//PR1006_REV_002685_TIMTRO
GVL.EF.S_Fus_1_01						:= GVL.IIVD.X_Fus_0_D1.v AND _FB_CanRx_Message_Unpack_261.S_Bit_6;
GVL.EF.S_Fus_1_02						:= GVL.IIVD.X_Fus_0_D1.v AND _FB_CanRx_Message_Unpack_261.S_Bit_4;
GVL.EF.S_Fus_1_03						:= GVL.IIVD.X_Fus_0_D1.v AND _FB_CanRx_Message_Unpack_261.S_Bit_2;
GVL.EF.S_Fus_1_04						:= GVL.IIVD.X_Fus_0_D1.v AND _FB_CanRx_Message_Unpack_261.S_Bit_0;	 
GVL.EF.S_Fus_1_05						:= GVL.IIVD.X_Fus_0_D2.v AND _FB_CanRx_Message_Unpack_261.S_Bit_14;
GVL.EF.S_Fus_1_06						:= GVL.IIVD.X_Fus_0_D2.v AND _FB_CanRx_Message_Unpack_261.S_Bit_12;
GVL.EF.S_Fus_1_07						:= GVL.IIVD.X_Fus_0_D2.v AND _FB_CanRx_Message_Unpack_261.S_Bit_10;
GVL.EF.S_Fus_1_08						:= GVL.IIVD.X_Fus_0_D2.v AND _FB_CanRx_Message_Unpack_261.S_Bit_8;					
GVL.EF.S_Fus_1_09						:= GVL.IIVD.X_Fus_0_D3.v AND _FB_CanRx_Message_Unpack_261.S_Bit_22;
GVL.EF.S_Fus_1_10						:= GVL.IIVD.X_Fus_0_D3.v AND _FB_CanRx_Message_Unpack_261.S_Bit_20;
GVL.EF.S_Fus_1_11						:= GVL.IIVD.X_Fus_0_D3.v AND _FB_CanRx_Message_Unpack_261.S_Bit_18;
GVL.EF.S_Fus_1_12						:= GVL.IIVD.X_Fus_0_D3.v AND _FB_CanRx_Message_Unpack_261.S_Bit_16;							  
GVL.EF.S_Fus_1_13						:= GVL.IIVD.X_Fus_0_D4.v AND _FB_CanRx_Message_Unpack_261.S_Bit_30;
GVL.EF.S_Fus_1_14						:= GVL.IIVD.X_Fus_0_D4.v AND _FB_CanRx_Message_Unpack_261.S_Bit_28;
GVL.EF.S_Fus_1_15						:= GVL.IIVD.X_Fus_0_D4.v AND _FB_CanRx_Message_Unpack_261.S_Bit_26;
GVL.EF.S_Fus_1_16						:= GVL.IIVD.X_Fus_0_D4.v AND _FB_CanRx_Message_Unpack_261.S_Bit_24;										
GVL.EF.S_Fus_1_17						:= GVL.IIVD.X_Fus_0_D5.v AND _FB_CanRx_Message_Unpack_261.S_Bit_38;
GVL.EF.S_Fus_1_18						:= GVL.IIVD.X_Fus_0_D5.v AND _FB_CanRx_Message_Unpack_261.S_Bit_36;
GVL.EF.S_Fus_1_19						:= GVL.IIVD.X_Fus_0_D5.v AND _FB_CanRx_Message_Unpack_261.S_Bit_34;
GVL.EF.S_Fus_1_20						:= GVL.IIVD.X_Fus_0_D5.v AND _FB_CanRx_Message_Unpack_261.S_Bit_32;		  
GVL.EF.S_Fus_1_21						:= GVL.IIVD.X_Fus_0_D6.v AND _FB_CanRx_Message_Unpack_261.S_Bit_46;
GVL.EF.S_Fus_1_22						:= GVL.IIVD.X_Fus_0_D6.v AND _FB_CanRx_Message_Unpack_261.S_Bit_44;
GVL.EF.S_Fus_1_23						:= GVL.IIVD.X_Fus_0_D6.v AND _FB_CanRx_Message_Unpack_261.S_Bit_42;
GVL.EF.S_Fus_1_24						:= GVL.IIVD.X_Fus_0_D6.v AND _FB_CanRx_Message_Unpack_261.S_Bit_40;		  
GVL.EF.S_Fus_1_25						:= GVL.IIVD.X_Fus_0_D7.v AND _FB_CanRx_Message_Unpack_261.S_Bit_54;
GVL.EF.S_Fus_1_26						:= GVL.IIVD.X_Fus_0_D7.v AND _FB_CanRx_Message_Unpack_261.S_Bit_52;
GVL.EF.S_Fus_1_27						:= GVL.IIVD.X_Fus_0_D7.v AND _FB_CanRx_Message_Unpack_261.S_Bit_50;
GVL.EF.S_Fus_1_28						:= GVL.IIVD.X_Fus_0_D7.v AND _FB_CanRx_Message_Unpack_261.S_Bit_48;												  
GVL.EF.S_Fus_1_29						:= GVL.IIVD.X_Fus_0_D8.v AND _FB_CanRx_Message_Unpack_261.S_Bit_62;
GVL.EF.S_Fus_1_30						:= GVL.IIVD.X_Fus_0_D8.v AND _FB_CanRx_Message_Unpack_261.S_Bit_60;
{endregion}
{endregion}

// PR1006_REV_002619_TIMTRO
{region " MESSAGE AREA :Sigorta_Kontrol_3- ID:262"}

_FB_CanRx_Message_Unpack_262 (		C_Enable	:= GVL.IIVD.S_CAN_Init,
     								Obj_CAN		:= ADR(GVL.IC.Obj_CAN0),
     								X_MsgID		:= 16#262,
     								Tm_MsgTmOut	:= TIME#2500MS,
     								S_Extended	:= 0,
     								S_ER_TmOut	=> GVL.IIVD.S_TmOut_Sigorta_Kontrol_3_0X262);

{region " SIGNAL AREA : NAME->X_Fus_2_D1 LENGTH->8 STARTBIT :0"}
Raw_X_Fus_2_D1							:= _FB_CanRx_Message_Unpack_262.X_Byte_7;
GVL.IIVD.X_Fus_2_D1.e					:= (Raw_X_Fus_2_D1 > 16#FD) AND (Raw_X_Fus_2_D1 < 16#FF);
GVL.IIVD.X_Fus_2_D1.na					:= (Raw_X_Fus_2_D1 = 16#FF);
GVL.IIVD.X_Fus_2_D1.RangeExcd			:= NOT (Raw_X_Fus_0_D1 >= 0) AND (Raw_X_Fus_2_D1 <= 254);
GVL.IIVD.X_Fus_2_D1.v					:= NOT( GVL.IIVD.S_TmOut_Sigorta_Kontrol_3_0X262 OR GVL.IIVD.X_Fus_2_D1.RangeExcd OR GVL.IIVD.X_Fus_2_D1.e OR GVL.IIVD.X_Fus_2_D1.na) ;
GVL.IIVD.X_Fus_2_D1.x					:= 
(*SELECT 1 : Is data valid ?*)				SEL(GVL.IIVD.X_Fus_2_D1.v,
(*DEFAULT value assigment*)					0,
(*Transmission is VALID*)					Raw_X_Fus_2_D1);

{endregion}
{region " SIGNAL AREA : NAME->X_Fus_2_D2 LENGTH->8 STARTBIT :8"}
Raw_X_Fus_2_D2							:= _FB_CanRx_Message_Unpack_262.X_Byte_6;
GVL.IIVD.X_Fus_2_D2.e					:= (Raw_X_Fus_2_D2 > 16#FD) AND (Raw_X_Fus_2_D2 < 16#FF);
GVL.IIVD.X_Fus_2_D2.na					:= (Raw_X_Fus_2_D2 = 16#FF);
GVL.IIVD.X_Fus_2_D2.RangeExcd			:= NOT (Raw_X_Fus_0_D1 >= 0) AND (Raw_X_Fus_2_D2 <= 254);
GVL.IIVD.X_Fus_2_D2.v					:= NOT( GVL.IIVD.S_TmOut_Sigorta_Kontrol_3_0X262 OR GVL.IIVD.X_Fus_2_D2.RangeExcd OR GVL.IIVD.X_Fus_2_D2.e OR GVL.IIVD.X_Fus_2_D2.na) ;
GVL.IIVD.X_Fus_2_D2.x					:= 
(*SELECT 1 : Is data valid ?*)				SEL(GVL.IIVD.X_Fus_2_D2.v,
(*DEFAULT value assigment*)					0,
(*Transmission is VALID*)					Raw_X_Fus_2_D2);

{endregion}
{region " SIGNAL AREA : NAME->X_Fus_2_D3 LENGTH->8 STARTBIT :16"}
Raw_X_Fus_2_D3							:= _FB_CanRx_Message_Unpack_262.X_Byte_5;
GVL.IIVD.X_Fus_2_D3.e					:= (Raw_X_Fus_2_D3 > 16#FD) AND (Raw_X_Fus_2_D3 < 16#FF);
GVL.IIVD.X_Fus_2_D3.na					:= (Raw_X_Fus_2_D3 = 16#FF);
GVL.IIVD.X_Fus_2_D3.RangeExcd			:= NOT (Raw_X_Fus_0_D1 >= 0) AND (Raw_X_Fus_2_D3 <= 254);
GVL.IIVD.X_Fus_2_D3.v					:= NOT( GVL.IIVD.S_TmOut_Sigorta_Kontrol_3_0X262 OR GVL.IIVD.X_Fus_2_D3.RangeExcd OR GVL.IIVD.X_Fus_2_D3.e OR GVL.IIVD.X_Fus_2_D3.na) ;
GVL.IIVD.X_Fus_2_D3.x					:= 
(*SELECT 1 : Is data valid ?*)				SEL(GVL.IIVD.X_Fus_2_D3.v,
(*DEFAULT value assigment*)					0,
(*Transmission is VALID*)					Raw_X_Fus_2_D3);

{endregion}
{region " SIGNAL AREA : NAME->X_Fus_2_D4 LENGTH->8 STARTBIT :24"}
Raw_X_Fus_2_D4							:= _FB_CanRx_Message_Unpack_262.X_Byte_4;
GVL.IIVD.X_Fus_2_D4.e					:= (Raw_X_Fus_2_D4 > 16#FD) AND (Raw_X_Fus_2_D4 < 16#FF);
GVL.IIVD.X_Fus_2_D4.na					:= (Raw_X_Fus_2_D4 = 16#FF);
GVL.IIVD.X_Fus_2_D4.RangeExcd			:= NOT (Raw_X_Fus_0_D1 >= 0) AND (Raw_X_Fus_2_D4 <= 254);
GVL.IIVD.X_Fus_2_D4.v					:= NOT( GVL.IIVD.S_TmOut_Sigorta_Kontrol_3_0X262 OR GVL.IIVD.X_Fus_2_D4.RangeExcd OR GVL.IIVD.X_Fus_2_D4.e OR GVL.IIVD.X_Fus_2_D4.na) ;
GVL.IIVD.X_Fus_2_D4.x					:= 
(*SELECT 1 : Is data valid ?*)				SEL(GVL.IIVD.X_Fus_2_D4.v,
(*DEFAULT value assigment*)					0,
(*Transmission is VALID*)					Raw_X_Fus_2_D4);

{endregion}
{region " SIGNAL AREA : NAME->X_Fus_2_D5 LENGTH->8 STARTBIT :32"}
Raw_X_Fus_2_D5							:= _FB_CanRx_Message_Unpack_262.X_Byte_3;
GVL.IIVD.X_Fus_2_D5.e					:= (Raw_X_Fus_2_D5 > 16#FD) AND (Raw_X_Fus_2_D5 < 16#FF);
GVL.IIVD.X_Fus_2_D5.na					:= (Raw_X_Fus_2_D5 = 16#FF);
GVL.IIVD.X_Fus_2_D5.RangeExcd			:= NOT (Raw_X_Fus_0_D1 >= 0) AND (Raw_X_Fus_2_D5 <= 254);
GVL.IIVD.X_Fus_2_D5.v					:= NOT( GVL.IIVD.S_TmOut_Sigorta_Kontrol_3_0X262 OR GVL.IIVD.X_Fus_2_D5.RangeExcd OR GVL.IIVD.X_Fus_2_D5.e OR GVL.IIVD.X_Fus_2_D5.na) ;
GVL.IIVD.X_Fus_2_D5.x					:= 
(*SELECT 1 : Is data valid ?*)				SEL(GVL.IIVD.X_Fus_2_D5.v,
(*DEFAULT value assigment*)					0,
(*Transmission is VALID*)					Raw_X_Fus_2_D5);

{endregion}
{region " SIGNAL AREA : NAME->X_Fus_2_D6 LENGTH->8 STARTBIT :40"}
Raw_X_Fus_2_D6							:= _FB_CanRx_Message_Unpack_262.X_Byte_2;
GVL.IIVD.X_Fus_2_D6.e					:= (Raw_X_Fus_2_D6 > 16#FD) AND (Raw_X_Fus_2_D6 < 16#FF);
GVL.IIVD.X_Fus_2_D6.na					:= (Raw_X_Fus_2_D6 = 16#FF);
GVL.IIVD.X_Fus_2_D6.RangeExcd			:= NOT (Raw_X_Fus_0_D1 >= 0) AND (Raw_X_Fus_2_D6 <= 254);
GVL.IIVD.X_Fus_2_D6.v					:= NOT( GVL.IIVD.S_TmOut_Sigorta_Kontrol_3_0X262 OR GVL.IIVD.X_Fus_2_D6.RangeExcd OR GVL.IIVD.X_Fus_2_D6.e OR GVL.IIVD.X_Fus_2_D6.na) ;
GVL.IIVD.X_Fus_2_D6.x					:= 
(*SELECT 1 : Is data valid ?*)				SEL(GVL.IIVD.X_Fus_2_D6.v,
(*DEFAULT value assigment*)					0,
(*Transmission is VALID*)					Raw_X_Fus_2_D6);

{endregion}
{region " SIGNAL AREA : NAME->X_Fus_2_D7 LENGTH->8 STARTBIT :48"}
Raw_X_Fus_2_D7							:= _FB_CanRx_Message_Unpack_262.X_Byte_1;
GVL.IIVD.X_Fus_2_D7.e					:= (Raw_X_Fus_2_D7 > 16#FD) AND (Raw_X_Fus_2_D7 < 16#FF);
GVL.IIVD.X_Fus_2_D7.na					:= (Raw_X_Fus_2_D7 = 16#FF);
GVL.IIVD.X_Fus_2_D7.RangeExcd			:= NOT (Raw_X_Fus_0_D1 >= 0) AND (Raw_X_Fus_2_D7 <= 254);
GVL.IIVD.X_Fus_2_D7.v					:= NOT( GVL.IIVD.S_TmOut_Sigorta_Kontrol_3_0X262 OR GVL.IIVD.X_Fus_2_D7.RangeExcd OR GVL.IIVD.X_Fus_2_D7.e OR GVL.IIVD.X_Fus_2_D7.na) ;
GVL.IIVD.X_Fus_2_D7.x					:= 
(*SELECT 1 : Is data valid ?*)				SEL(GVL.IIVD.X_Fus_2_D7.v,
(*DEFAULT value assigment*)					0,
(*Transmission is VALID*)					Raw_X_Fus_2_D7);

{endregion}
{region " SIGNAL AREA : NAME->X_Fus_2_D8 LENGTH->8 STARTBIT :56"}
Raw_X_Fus_2_D8							:= _FB_CanRx_Message_Unpack_262.X_Byte_0;
GVL.IIVD.X_Fus_2_D8.e					:= (Raw_X_Fus_2_D8 > 16#FD) AND (Raw_X_Fus_2_D8 < 16#FF);
GVL.IIVD.X_Fus_2_D8.na					:= (Raw_X_Fus_2_D8 = 16#FF);
GVL.IIVD.X_Fus_2_D8.RangeExcd			:= NOT (Raw_X_Fus_0_D1 >= 0) AND (Raw_X_Fus_2_D8 <= 254);
GVL.IIVD.X_Fus_2_D8.v					:= NOT( GVL.IIVD.S_TmOut_Sigorta_Kontrol_3_0X262 OR GVL.IIVD.X_Fus_2_D8.RangeExcd OR GVL.IIVD.X_Fus_2_D8.e OR GVL.IIVD.X_Fus_2_D8.na) ;
GVL.IIVD.X_Fus_2_D8.x					:= 
(*SELECT 1 : Is data valid ?*)				SEL(GVL.IIVD.X_Fus_2_D8.v,
(*DEFAULT value assigment*)					0,
(*Transmission is VALID*)					Raw_X_Fus_2_D8);

//PR1006_REV_002685_TIMTRO
GVL.EF.S_Fus_2_01						:= GVL.IIVD.X_Fus_0_D1.v AND _FB_CanRx_Message_Unpack_262.S_Bit_6;
GVL.EF.S_Fus_2_02						:= GVL.IIVD.X_Fus_0_D1.v AND _FB_CanRx_Message_Unpack_262.S_Bit_4;
GVL.EF.S_Fus_2_03						:= GVL.IIVD.X_Fus_0_D1.v AND _FB_CanRx_Message_Unpack_262.S_Bit_2;
GVL.EF.S_Fus_2_04						:= GVL.IIVD.X_Fus_0_D1.v AND _FB_CanRx_Message_Unpack_262.S_Bit_0;	  
GVL.EF.S_Fus_2_05						:= GVL.IIVD.X_Fus_0_D2.v AND _FB_CanRx_Message_Unpack_262.S_Bit_14;
GVL.EF.S_Fus_2_06						:= GVL.IIVD.X_Fus_0_D2.v AND _FB_CanRx_Message_Unpack_262.S_Bit_12;
GVL.EF.S_Fus_2_07						:= GVL.IIVD.X_Fus_0_D2.v AND _FB_CanRx_Message_Unpack_262.S_Bit_10;
GVL.EF.S_Fus_2_08						:= GVL.IIVD.X_Fus_0_D2.v AND _FB_CanRx_Message_Unpack_262.S_Bit_8;					
GVL.EF.S_Fus_2_09						:= GVL.IIVD.X_Fus_0_D3.v AND _FB_CanRx_Message_Unpack_262.S_Bit_22;
GVL.EF.S_Fus_2_10						:= GVL.IIVD.X_Fus_0_D3.v AND _FB_CanRx_Message_Unpack_262.S_Bit_20;
GVL.EF.S_Fus_2_11						:= GVL.IIVD.X_Fus_0_D3.v AND _FB_CanRx_Message_Unpack_262.S_Bit_18;
GVL.EF.S_Fus_2_12						:= GVL.IIVD.X_Fus_0_D3.v AND _FB_CanRx_Message_Unpack_262.S_Bit_16;							  
GVL.EF.S_Fus_2_13						:= GVL.IIVD.X_Fus_0_D4.v AND _FB_CanRx_Message_Unpack_262.S_Bit_30;
GVL.EF.S_Fus_2_14						:= GVL.IIVD.X_Fus_0_D4.v AND _FB_CanRx_Message_Unpack_262.S_Bit_28;
GVL.EF.S_Fus_2_15						:= GVL.IIVD.X_Fus_0_D4.v AND _FB_CanRx_Message_Unpack_262.S_Bit_26;
GVL.EF.S_Fus_2_16						:= GVL.IIVD.X_Fus_0_D4.v AND _FB_CanRx_Message_Unpack_262.S_Bit_24;										
GVL.EF.S_Fus_2_17						:= GVL.IIVD.X_Fus_0_D5.v AND _FB_CanRx_Message_Unpack_262.S_Bit_38;
GVL.EF.S_Fus_2_18						:= GVL.IIVD.X_Fus_0_D5.v AND _FB_CanRx_Message_Unpack_262.S_Bit_36;
GVL.EF.S_Fus_2_19						:= GVL.IIVD.X_Fus_0_D5.v AND _FB_CanRx_Message_Unpack_262.S_Bit_34;
GVL.EF.S_Fus_2_20						:= GVL.IIVD.X_Fus_0_D5.v AND _FB_CanRx_Message_Unpack_262.S_Bit_32;		  
GVL.EF.S_Fus_2_21						:= GVL.IIVD.X_Fus_0_D6.v AND _FB_CanRx_Message_Unpack_262.S_Bit_46;
GVL.EF.S_Fus_2_22						:= GVL.IIVD.X_Fus_0_D6.v AND _FB_CanRx_Message_Unpack_262.S_Bit_44;
GVL.EF.S_Fus_2_23						:= GVL.IIVD.X_Fus_0_D6.v AND _FB_CanRx_Message_Unpack_262.S_Bit_42;
GVL.EF.S_Fus_2_24						:= GVL.IIVD.X_Fus_0_D6.v AND _FB_CanRx_Message_Unpack_262.S_Bit_40;		  
GVL.EF.S_Fus_2_25						:= GVL.IIVD.X_Fus_0_D7.v AND _FB_CanRx_Message_Unpack_262.S_Bit_54;
GVL.EF.S_Fus_2_26						:= GVL.IIVD.X_Fus_0_D7.v AND _FB_CanRx_Message_Unpack_262.S_Bit_52;
GVL.EF.S_Fus_2_27						:= GVL.IIVD.X_Fus_0_D7.v AND _FB_CanRx_Message_Unpack_262.S_Bit_50;
GVL.EF.S_Fus_2_28						:= GVL.IIVD.X_Fus_0_D7.v AND _FB_CanRx_Message_Unpack_262.S_Bit_48;												  
GVL.EF.S_Fus_2_29						:= GVL.IIVD.X_Fus_0_D8.v AND _FB_CanRx_Message_Unpack_262.S_Bit_62;
GVL.EF.S_Fus_2_30						:= GVL.IIVD.X_Fus_0_D8.v AND _FB_CanRx_Message_Unpack_262.S_Bit_60;
{endregion}
{endregion}

{region " MESSAGE AREA :Parametre_1- ID:263"}

_FB_CanRx_Message_Unpack_263 (		C_Enable	:= GVL.IIVD.S_CAN_Init,
     								Obj_CAN		:= ADR(GVL.IC.Obj_CAN0),
     								X_MsgID		:= 16#263,
     								Tm_MsgTmOut	:= TIME#2500MS,
     								S_Extended	:= 0,
     								S_ER_TmOut	=> GVL.IIVD.S_TmOut_Parametre_1_0X263);

{region " SIGNAL AREA : NAME->C_Param_Set LENGTH->2 STARTBIT :0"}
GVL.IIVD.C_Param_Set.v					:= NOT GVL.IIVD.S_TmOut_Parametre_1_0X263 AND NOT _FB_CanRx_Message_Unpack_263.S_Bit_1;
GVL.IIVD.C_Param_Set.x					:= GVL.IIVD.C_Param_Set.v AND _FB_CanRx_Message_Unpack_263.S_Bit_0;
GVL.IIVD.C_Param_Set.e					:= _FB_CanRx_Message_Unpack_263.S_Bit_1 AND NOT _FB_CanRx_Message_Unpack_263.S_Bit_0 ;
GVL.IIVD.C_Param_Set.na					:= _FB_CanRx_Message_Unpack_263.S_Bit_1 AND _FB_CanRx_Message_Unpack_263.S_Bit_0 ;
{endregion}	 	 
{region " SIGNAL AREA : NAME->P_Set_Tm_Dr_Cl_Rls LENGTH->8 STARTBIT :8"}
Raw_P_Set_Tm_Dr_Cl_Rls					:= _FB_CanRx_Message_Unpack_263.X_Byte_1;
GVL.IIVD.P_Set_Tm_Dr_Cl_Rls.e			:= (Raw_P_Set_Tm_Dr_Cl_Rls > 16#FD) AND (Raw_P_Set_Tm_Dr_Cl_Rls < 16#FF);
GVL.IIVD.P_Set_Tm_Dr_Cl_Rls.na			:= (Raw_P_Set_Tm_Dr_Cl_Rls = 16#FF);
GVL.IIVD.P_Set_Tm_Dr_Cl_Rls.RangeExcd	:= NOT ((USINT_TO_REAL(BYTE_TO_USINT(Raw_P_Set_Tm_Dr_Cl_Rls)) >= 0) AND (USINT_TO_REAL(BYTE_TO_USINT(Raw_P_Set_Tm_Dr_Cl_Rls)) <= 250));
GVL.IIVD.P_Set_Tm_Dr_Cl_Rls.v			:= NOT( GVL.IIVD.S_TmOut_Parametre_1_0X263 OR GVL.IIVD.P_Set_Tm_Dr_Cl_Rls.RangeExcd OR GVL.IIVD.P_Set_Tm_Dr_Cl_Rls.e OR GVL.IIVD.P_Set_Tm_Dr_Cl_Rls.na) ;
GVL.IIVD.P_Set_Tm_Dr_Cl_Rls.x			:= 
(*SELECT 1 : Is data valid ?*)				SEL(GVL.IIVD.P_Set_Tm_Dr_Cl_Rls.v,
(*DEFAULT value assigment*)					0,
(*Transmission is VALID*)					USINT_TO_REAL(BYTE_TO_USINT(Raw_P_Set_Tm_Dr_Cl_Rls)) * 5);	 //PR1006_REV_002664_TIMTRO
{endregion}	 	
{region " SIGNAL AREA : NAME->P_Set_Tm_Rout_Pnl_ShtDn LENGTH->8 STARTBIT :16"}
Raw_P_Set_Tm_Rout_Pnl_ShtDn					:= _FB_CanRx_Message_Unpack_263.X_Byte_2;
GVL.IIVD.P_Set_Tm_Rout_Pnl_ShtDn.e			:= (Raw_P_Set_Tm_Rout_Pnl_ShtDn > 16#FD) AND (Raw_P_Set_Tm_Rout_Pnl_ShtDn < 16#FF);
GVL.IIVD.P_Set_Tm_Rout_Pnl_ShtDn.na			:= (Raw_P_Set_Tm_Rout_Pnl_ShtDn = 16#FF);
GVL.IIVD.P_Set_Tm_Rout_Pnl_ShtDn.RangeExcd	:= NOT ((USINT_TO_REAL(BYTE_TO_USINT(Raw_P_Set_Tm_Rout_Pnl_ShtDn)) >= 0) AND (USINT_TO_REAL(BYTE_TO_USINT(Raw_P_Set_Tm_Rout_Pnl_ShtDn)) <= 250));
GVL.IIVD.P_Set_Tm_Rout_Pnl_ShtDn.v			:= NOT( GVL.IIVD.S_TmOut_Parametre_1_0X263 OR GVL.IIVD.P_Set_Tm_Rout_Pnl_ShtDn.RangeExcd OR GVL.IIVD.P_Set_Tm_Rout_Pnl_ShtDn.e OR GVL.IIVD.P_Set_Tm_Rout_Pnl_ShtDn.na) ;
GVL.IIVD.P_Set_Tm_Rout_Pnl_ShtDn.x			:= 
(*SELECT 1 : Is data valid ?*)				SEL(GVL.IIVD.P_Set_Tm_Rout_Pnl_ShtDn.v,
(*DEFAULT value assigment*)					0,
(*Transmission is VALID*)					USINT_TO_REAL(BYTE_TO_USINT(Raw_P_Set_Tm_Rout_Pnl_ShtDn)) * 5);	  	//PR1006_REV_002664_TIMTRO
{endregion}	 
{region " SIGNAL AREA : NAME->P_Set_Tm_Lgt_Dr_ShtDn LENGTH->8 STARTBIT :24"}
Raw_P_Set_Tm_Lgt_Dr_ShtDn					:= _FB_CanRx_Message_Unpack_263.X_Byte_3;
GVL.IIVD.P_Set_Tm_Lgt_Dr_ShtDn.e			:= (Raw_P_Set_Tm_Lgt_Dr_ShtDn > 16#FD) AND (Raw_P_Set_Tm_Lgt_Dr_ShtDn < 16#FF);
GVL.IIVD.P_Set_Tm_Lgt_Dr_ShtDn.na			:= (Raw_P_Set_Tm_Lgt_Dr_ShtDn = 16#FF);
GVL.IIVD.P_Set_Tm_Lgt_Dr_ShtDn.RangeExcd	:= NOT ((USINT_TO_REAL(BYTE_TO_USINT(Raw_P_Set_Tm_Lgt_Dr_ShtDn)) >= 0) AND (USINT_TO_REAL(BYTE_TO_USINT(Raw_P_Set_Tm_Lgt_Dr_ShtDn)) <= 250));
GVL.IIVD.P_Set_Tm_Lgt_Dr_ShtDn.v			:= NOT( GVL.IIVD.S_TmOut_Parametre_1_0X263 OR GVL.IIVD.P_Set_Tm_Lgt_Dr_ShtDn.RangeExcd OR GVL.IIVD.P_Set_Tm_Lgt_Dr_ShtDn.e OR GVL.IIVD.P_Set_Tm_Lgt_Dr_ShtDn.na) ;
GVL.IIVD.P_Set_Tm_Lgt_Dr_ShtDn.x			:= 
(*SELECT 1 : Is data valid ?*)					SEL(GVL.IIVD.P_Set_Tm_Lgt_Dr_ShtDn.v,
(*DEFAULT value assigment*)						0,
(*Transmission is VALID*)						USINT_TO_REAL(BYTE_TO_USINT(Raw_P_Set_Tm_Lgt_Dr_ShtDn)) * 5);	 //PR1006_REV_002664_TIMTRO 
{endregion}	 		
{endregion}	 	  

// PR1006_REV_002619_TIMTRO
{region " MESSAGE AREA :Sigorta_Kontrol_4- ID:264"}

_FB_CanRx_Message_Unpack_264 (		C_Enable	:= GVL.IIVD.S_CAN_Init,
     								Obj_CAN		:= ADR(GVL.IC.Obj_CAN0),
     								X_MsgID		:= 16#264,
     								Tm_MsgTmOut	:= TIME#2500MS,
     								S_Extended	:= 0,
     								S_ER_TmOut	=> GVL.IIVD.S_TmOut_Sigorta_Kontrol_4_0X264);

{region " SIGNAL AREA : NAME->X_Fus_3_D1 LENGTH->8 STARTBIT :0"}
Raw_X_Fus_3_D1							:= _FB_CanRx_Message_Unpack_264.X_Byte_7;
GVL.IIVD.X_Fus_3_D1.e					:= (Raw_X_Fus_3_D1 > 16#FD) AND (Raw_X_Fus_3_D1 < 16#FF);
GVL.IIVD.X_Fus_3_D1.na					:= (Raw_X_Fus_3_D1 = 16#FF);
GVL.IIVD.X_Fus_3_D1.RangeExcd			:= NOT (Raw_X_Fus_0_D1 >= 0) AND (Raw_X_Fus_3_D1 <= 254);
GVL.IIVD.X_Fus_3_D1.v					:= NOT( GVL.IIVD.S_TmOut_Sigorta_Kontrol_4_0X264 OR GVL.IIVD.X_Fus_3_D1.RangeExcd OR GVL.IIVD.X_Fus_3_D1.e OR GVL.IIVD.X_Fus_3_D1.na) ;
GVL.IIVD.X_Fus_3_D1.x					:= 
(*SELECT 1 : Is data valid ?*)				SEL(GVL.IIVD.X_Fus_3_D1.v,
(*DEFAULT value assigment*)					0,
(*Transmission is VALID*)					Raw_X_Fus_3_D1);

{endregion}
{region " SIGNAL AREA : NAME->X_Fus_3_D2 LENGTH->8 STARTBIT :8"}
Raw_X_Fus_3_D2							:= _FB_CanRx_Message_Unpack_264.X_Byte_6;
GVL.IIVD.X_Fus_3_D2.e					:= (Raw_X_Fus_3_D2 > 16#FD) AND (Raw_X_Fus_3_D2 < 16#FF);
GVL.IIVD.X_Fus_3_D2.na					:= (Raw_X_Fus_3_D2 = 16#FF);
GVL.IIVD.X_Fus_3_D2.RangeExcd			:= NOT (Raw_X_Fus_0_D1 >= 0) AND (Raw_X_Fus_3_D2 <= 254);
GVL.IIVD.X_Fus_3_D2.v					:= NOT( GVL.IIVD.S_TmOut_Sigorta_Kontrol_4_0X264 OR GVL.IIVD.X_Fus_3_D2.RangeExcd OR GVL.IIVD.X_Fus_3_D2.e OR GVL.IIVD.X_Fus_3_D2.na) ;
GVL.IIVD.X_Fus_3_D2.x					:= 
(*SELECT 1 : Is data valid ?*)				SEL(GVL.IIVD.X_Fus_3_D2.v,
(*DEFAULT value assigment*)					0,
(*Transmission is VALID*)					Raw_X_Fus_3_D2);

{endregion}
{region " SIGNAL AREA : NAME->X_Fus_3_D3 LENGTH->8 STARTBIT :16"}
Raw_X_Fus_3_D3							:= _FB_CanRx_Message_Unpack_264.X_Byte_5;
GVL.IIVD.X_Fus_3_D3.e					:= (Raw_X_Fus_3_D3 > 16#FD) AND (Raw_X_Fus_3_D3 < 16#FF);
GVL.IIVD.X_Fus_3_D3.na					:= (Raw_X_Fus_3_D3 = 16#FF);
GVL.IIVD.X_Fus_3_D3.RangeExcd			:= NOT (Raw_X_Fus_0_D1 >= 0) AND (Raw_X_Fus_3_D3 <= 254);
GVL.IIVD.X_Fus_3_D3.v					:= NOT( GVL.IIVD.S_TmOut_Sigorta_Kontrol_4_0X264 OR GVL.IIVD.X_Fus_3_D3.RangeExcd OR GVL.IIVD.X_Fus_3_D3.e OR GVL.IIVD.X_Fus_3_D3.na) ;
GVL.IIVD.X_Fus_3_D3.x					:= 
(*SELECT 1 : Is data valid ?*)				SEL(GVL.IIVD.X_Fus_3_D3.v,
(*DEFAULT value assigment*)					0,
(*Transmission is VALID*)					Raw_X_Fus_3_D3);

{endregion}
{region " SIGNAL AREA : NAME->X_Fus_3_D4 LENGTH->8 STARTBIT :24"}
Raw_X_Fus_3_D4							:= _FB_CanRx_Message_Unpack_264.X_Byte_4;
GVL.IIVD.X_Fus_3_D4.e					:= (Raw_X_Fus_3_D4 > 16#FD) AND (Raw_X_Fus_3_D4 < 16#FF);
GVL.IIVD.X_Fus_3_D4.na					:= (Raw_X_Fus_3_D4 = 16#FF);
GVL.IIVD.X_Fus_3_D4.RangeExcd			:= NOT (Raw_X_Fus_0_D1 >= 0) AND (Raw_X_Fus_3_D4 <= 254);
GVL.IIVD.X_Fus_3_D4.v					:= NOT( GVL.IIVD.S_TmOut_Sigorta_Kontrol_4_0X264 OR GVL.IIVD.X_Fus_3_D4.RangeExcd OR GVL.IIVD.X_Fus_3_D4.e OR GVL.IIVD.X_Fus_3_D4.na) ;
GVL.IIVD.X_Fus_3_D4.x					:= 
(*SELECT 1 : Is data valid ?*)				SEL(GVL.IIVD.X_Fus_3_D4.v,
(*DEFAULT value assigment*)					0,
(*Transmission is VALID*)					Raw_X_Fus_3_D4);

{endregion}
{region " SIGNAL AREA : NAME->X_Fus_3_D5 LENGTH->8 STARTBIT :32"}
Raw_X_Fus_3_D5							:= _FB_CanRx_Message_Unpack_264.X_Byte_3;
GVL.IIVD.X_Fus_3_D5.e					:= (Raw_X_Fus_3_D5 > 16#FD) AND (Raw_X_Fus_3_D5 < 16#FF);
GVL.IIVD.X_Fus_3_D5.na					:= (Raw_X_Fus_3_D5 = 16#FF);
GVL.IIVD.X_Fus_3_D5.RangeExcd			:= NOT (Raw_X_Fus_0_D1 >= 0) AND (Raw_X_Fus_3_D5 <= 254);
GVL.IIVD.X_Fus_3_D5.v					:= NOT( GVL.IIVD.S_TmOut_Sigorta_Kontrol_4_0X264 OR GVL.IIVD.X_Fus_3_D5.RangeExcd OR GVL.IIVD.X_Fus_3_D5.e OR GVL.IIVD.X_Fus_3_D5.na) ;
GVL.IIVD.X_Fus_3_D5.x					:= 
(*SELECT 1 : Is data valid ?*)				SEL(GVL.IIVD.X_Fus_3_D5.v,
(*DEFAULT value assigment*)					0,
(*Transmission is VALID*)					Raw_X_Fus_3_D5);

{endregion}
{region " SIGNAL AREA : NAME->X_Fus_3_D6 LENGTH->8 STARTBIT :40"}
Raw_X_Fus_3_D6							:= _FB_CanRx_Message_Unpack_264.X_Byte_2;
GVL.IIVD.X_Fus_3_D6.e					:= (Raw_X_Fus_3_D6 > 16#FD) AND (Raw_X_Fus_3_D6 < 16#FF);
GVL.IIVD.X_Fus_3_D6.na					:= (Raw_X_Fus_3_D6 = 16#FF);
GVL.IIVD.X_Fus_3_D6.RangeExcd			:= NOT (Raw_X_Fus_0_D1 >= 0) AND (Raw_X_Fus_3_D6 <= 254);
GVL.IIVD.X_Fus_3_D6.v					:= NOT( GVL.IIVD.S_TmOut_Sigorta_Kontrol_4_0X264 OR GVL.IIVD.X_Fus_3_D6.RangeExcd OR GVL.IIVD.X_Fus_3_D6.e OR GVL.IIVD.X_Fus_3_D6.na) ;
GVL.IIVD.X_Fus_3_D6.x					:= 
(*SELECT 1 : Is data valid ?*)				SEL(GVL.IIVD.X_Fus_3_D6.v,
(*DEFAULT value assigment*)					0,
(*Transmission is VALID*)					Raw_X_Fus_3_D6);

{endregion}
{region " SIGNAL AREA : NAME->X_Fus_3_D7 LENGTH->8 STARTBIT :48"}
Raw_X_Fus_3_D7							:= _FB_CanRx_Message_Unpack_264.X_Byte_1;
GVL.IIVD.X_Fus_3_D7.e					:= (Raw_X_Fus_3_D7 > 16#FD) AND (Raw_X_Fus_3_D7 < 16#FF);
GVL.IIVD.X_Fus_3_D7.na					:= (Raw_X_Fus_3_D7 = 16#FF);
GVL.IIVD.X_Fus_3_D7.RangeExcd			:= NOT (Raw_X_Fus_0_D1 >= 0) AND (Raw_X_Fus_3_D7 <= 254);
GVL.IIVD.X_Fus_3_D7.v					:= NOT( GVL.IIVD.S_TmOut_Sigorta_Kontrol_4_0X264 OR GVL.IIVD.X_Fus_3_D7.RangeExcd OR GVL.IIVD.X_Fus_3_D7.e OR GVL.IIVD.X_Fus_3_D7.na) ;
GVL.IIVD.X_Fus_3_D7.x					:= 
(*SELECT 1 : Is data valid ?*)				SEL(GVL.IIVD.X_Fus_3_D7.v,
(*DEFAULT value assigment*)					0,
(*Transmission is VALID*)					Raw_X_Fus_3_D7);

{endregion}
{region " SIGNAL AREA : NAME->X_Fus_3_D8 LENGTH->8 STARTBIT :56"}
Raw_X_Fus_3_D8							:= _FB_CanRx_Message_Unpack_264.X_Byte_0;
GVL.IIVD.X_Fus_3_D8.e					:= (Raw_X_Fus_3_D8 > 16#FD) AND (Raw_X_Fus_3_D8 < 16#FF);
GVL.IIVD.X_Fus_3_D8.na					:= (Raw_X_Fus_3_D8 = 16#FF);
GVL.IIVD.X_Fus_3_D8.RangeExcd			:= NOT (Raw_X_Fus_0_D1 >= 0) AND (Raw_X_Fus_3_D8 <= 254);
GVL.IIVD.X_Fus_3_D8.v					:= NOT( GVL.IIVD.S_TmOut_Sigorta_Kontrol_4_0X264 OR GVL.IIVD.X_Fus_3_D8.RangeExcd OR GVL.IIVD.X_Fus_3_D8.e OR GVL.IIVD.X_Fus_3_D8.na) ;
GVL.IIVD.X_Fus_3_D8.x					:= 
(*SELECT 1 : Is data valid ?*)				SEL(GVL.IIVD.X_Fus_3_D8.v,
(*DEFAULT value assigment*)					0,
(*Transmission is VALID*)					Raw_X_Fus_3_D8);

//PR1006_REV_002685_TIMTRO
GVL.EF.S_Fus_3_01						:= GVL.IIVD.X_Fus_0_D1.v AND _FB_CanRx_Message_Unpack_264.S_Bit_6;
GVL.EF.S_Fus_3_02						:= GVL.IIVD.X_Fus_0_D1.v AND _FB_CanRx_Message_Unpack_264.S_Bit_4;
GVL.EF.S_Fus_3_03						:= GVL.IIVD.X_Fus_0_D1.v AND _FB_CanRx_Message_Unpack_264.S_Bit_2;
GVL.EF.S_Fus_3_04						:= GVL.IIVD.X_Fus_0_D1.v AND _FB_CanRx_Message_Unpack_264.S_Bit_0;	  
GVL.EF.S_Fus_3_05						:= GVL.IIVD.X_Fus_0_D2.v AND _FB_CanRx_Message_Unpack_264.S_Bit_14;
GVL.EF.S_Fus_3_06						:= GVL.IIVD.X_Fus_0_D2.v AND _FB_CanRx_Message_Unpack_264.S_Bit_12;
GVL.EF.S_Fus_3_07						:= GVL.IIVD.X_Fus_0_D2.v AND _FB_CanRx_Message_Unpack_264.S_Bit_10;
GVL.EF.S_Fus_3_08						:= GVL.IIVD.X_Fus_0_D2.v AND _FB_CanRx_Message_Unpack_264.S_Bit_8;					
GVL.EF.S_Fus_3_09						:= GVL.IIVD.X_Fus_0_D3.v AND _FB_CanRx_Message_Unpack_264.S_Bit_22;
GVL.EF.S_Fus_3_10						:= GVL.IIVD.X_Fus_0_D3.v AND _FB_CanRx_Message_Unpack_264.S_Bit_20;
GVL.EF.S_Fus_3_11						:= GVL.IIVD.X_Fus_0_D3.v AND _FB_CanRx_Message_Unpack_264.S_Bit_18;
GVL.EF.S_Fus_3_12						:= GVL.IIVD.X_Fus_0_D3.v AND _FB_CanRx_Message_Unpack_264.S_Bit_16;							  
GVL.EF.S_Fus_3_13						:= GVL.IIVD.X_Fus_0_D4.v AND _FB_CanRx_Message_Unpack_264.S_Bit_30;
GVL.EF.S_Fus_3_14						:= GVL.IIVD.X_Fus_0_D4.v AND _FB_CanRx_Message_Unpack_264.S_Bit_28;
GVL.EF.S_Fus_3_15						:= GVL.IIVD.X_Fus_0_D4.v AND _FB_CanRx_Message_Unpack_264.S_Bit_26;
GVL.EF.S_Fus_3_16						:= GVL.IIVD.X_Fus_0_D4.v AND _FB_CanRx_Message_Unpack_264.S_Bit_24;										
GVL.EF.S_Fus_3_17						:= GVL.IIVD.X_Fus_0_D5.v AND _FB_CanRx_Message_Unpack_264.S_Bit_38;
GVL.EF.S_Fus_3_18						:= GVL.IIVD.X_Fus_0_D5.v AND _FB_CanRx_Message_Unpack_264.S_Bit_36;
GVL.EF.S_Fus_3_19						:= GVL.IIVD.X_Fus_0_D5.v AND _FB_CanRx_Message_Unpack_264.S_Bit_34;
GVL.EF.S_Fus_3_20						:= GVL.IIVD.X_Fus_0_D5.v AND _FB_CanRx_Message_Unpack_264.S_Bit_32;		  
GVL.EF.S_Fus_3_21						:= GVL.IIVD.X_Fus_0_D6.v AND _FB_CanRx_Message_Unpack_264.S_Bit_46;
GVL.EF.S_Fus_3_22						:= GVL.IIVD.X_Fus_0_D6.v AND _FB_CanRx_Message_Unpack_264.S_Bit_44;
GVL.EF.S_Fus_3_23						:= GVL.IIVD.X_Fus_0_D6.v AND _FB_CanRx_Message_Unpack_264.S_Bit_42;
GVL.EF.S_Fus_3_24						:= GVL.IIVD.X_Fus_0_D6.v AND _FB_CanRx_Message_Unpack_264.S_Bit_40;		  
GVL.EF.S_Fus_3_25						:= GVL.IIVD.X_Fus_0_D7.v AND _FB_CanRx_Message_Unpack_264.S_Bit_54;
GVL.EF.S_Fus_3_26						:= GVL.IIVD.X_Fus_0_D7.v AND _FB_CanRx_Message_Unpack_264.S_Bit_52;
GVL.EF.S_Fus_3_27						:= GVL.IIVD.X_Fus_0_D7.v AND _FB_CanRx_Message_Unpack_264.S_Bit_50;
GVL.EF.S_Fus_3_28						:= GVL.IIVD.X_Fus_0_D7.v AND _FB_CanRx_Message_Unpack_264.S_Bit_48;												  
GVL.EF.S_Fus_3_29						:= GVL.IIVD.X_Fus_0_D8.v AND _FB_CanRx_Message_Unpack_264.S_Bit_62;
GVL.EF.S_Fus_3_30						:= GVL.IIVD.X_Fus_0_D8.v AND _FB_CanRx_Message_Unpack_264.S_Bit_60;			   
{endregion}
{endregion}

// PR1006_SRS_000531_TIMTRO 
{region " MESSAGE AREA : Vehicle_Info_2 - ID:2E1"}

_FB_CanRx_Message_Unpack_2E1 (		C_Enable	:= GVL.IIVD.S_CAN_Init,
     								Obj_CAN		:= ADR(GVL.IC.Obj_CAN0),
     								X_MsgID		:= 16#2E1,
     								Tm_MsgTmOut	:= TIME#10000MS,
     								S_Extended	:= 0,
     								S_ER_TmOut	=> GVL.IIVD.S_TmOut_Arac_Bilgi_2_0X2E1);

{region " SIGNAL AREA : NAME->X_Sw_Ver_Mjr_DWP LENGTH->8 STARTBIT :0"}
Raw_X_Sw_Ver_Mjr_DWP						:= _FB_CanRx_Message_Unpack_2E1.X_Byte_0;
GVL.IIVD.X_Sw_Ver_Mjr_DWP.e					:= (Raw_X_Sw_Ver_Mjr_DWP > 16#FD) AND (Raw_X_Sw_Ver_Mjr_DWP < 16#FF);
GVL.IIVD.X_Sw_Ver_Mjr_DWP.na				:= (Raw_X_Sw_Ver_Mjr_DWP = 16#FF);
GVL.IIVD.X_Sw_Ver_Mjr_DWP.RangeExcd			:= NOT ((USINT_TO_REAL(BYTE_TO_USINT(Raw_X_Sw_Ver_Mjr_DWP)) >= 0) AND (USINT_TO_REAL(BYTE_TO_USINT(Raw_X_Sw_Ver_Mjr_DWP)) <= 250));
GVL.IIVD.X_Sw_Ver_Mjr_DWP.v					:= NOT( GVL.IIVD.S_TmOut_Arac_Bilgi_2_0X2E1 OR GVL.IIVD.X_Sw_Ver_Mjr_DWP.RangeExcd OR GVL.IIVD.X_Sw_Ver_Mjr_DWP.e OR GVL.IIVD.X_Sw_Ver_Mjr_DWP.na);
GVL.IIVD.X_Sw_Ver_Mjr_DWP.x					:= 
(*SELECT 1 : Is data valid ?*)					SEL(GVL.IIVD.X_Sw_Ver_Mjr_DWP.v,
(*DEFAULT value assigment*)						0,
(*Transmission is VALID*)						USINT_TO_REAL(BYTE_TO_USINT(Raw_X_Sw_Ver_Mjr_DWP)));	
{endregion}
		  
{region SIGNAL AREA: NAME->X_Sw_Ver_Mnr_DWP LENGTH->8 STARTBIT:8}
Raw_X_Sw_Ver_Mnr_DWP						:= _FB_CanRx_Message_Unpack_2E1.X_Byte_1;
GVL.IIVD.X_Sw_Ver_Mnr_DWP.e					:= (Raw_X_Sw_Ver_Mnr_DWP > 16#FD) AND (Raw_X_Sw_Ver_Mnr_DWP < 16#FF);
GVL.IIVD.X_Sw_Ver_Mnr_DWP.na				:= (Raw_X_Sw_Ver_Mnr_DWP = 16#FF);
GVL.IIVD.X_Sw_Ver_Mnr_DWP.RangeExcd			:= NOT ((USINT_TO_REAL(BYTE_TO_USINT(Raw_X_Sw_Ver_Mnr_DWP)) >= 0) AND (USINT_TO_REAL(BYTE_TO_USINT(Raw_X_Sw_Ver_Mnr_DWP)) <= 250));
GVL.IIVD.X_Sw_Ver_Mnr_DWP.v					:= NOT( GVL.IIVD.S_TmOut_Arac_Bilgi_2_0X2E1 OR GVL.IIVD.X_Sw_Ver_Mnr_DWP.RangeExcd OR GVL.IIVD.X_Sw_Ver_Mnr_DWP.e OR GVL.IIVD.X_Sw_Ver_Mnr_DWP.na) ;
GVL.IIVD.X_Sw_Ver_Mnr_DWP.x					:= 
(*SELECT 1 : Is data valid ?*)					SEL(GVL.IIVD.X_Sw_Ver_Mnr_DWP.v,
(*DEFAULT value assigment*)						0,
(*Transmission is VALID*)						USINT_TO_REAL(BYTE_TO_USINT(Raw_X_Sw_Ver_Mnr_DWP)));	
{endregion}
		  
{region " SIGNAL AREA : NAME->X_Sw_Ver_Tst_DWP LENGTH->8 STARTBIT :16"}
Raw_X_Sw_Ver_Tst_DWP						:= _FB_CanRx_Message_Unpack_2E1.X_Byte_2;
GVL.IIVD.X_Sw_Ver_Tst_DWP.e					:= (Raw_X_Sw_Ver_Tst_DWP > 16#FD) AND (Raw_X_Sw_Ver_Tst_DWP < 16#FF);
GVL.IIVD.X_Sw_Ver_Tst_DWP.na				:= (Raw_X_Sw_Ver_Tst_DWP = 16#FF);
GVL.IIVD.X_Sw_Ver_Tst_DWP.RangeExcd			:= NOT ((USINT_TO_REAL(BYTE_TO_USINT(Raw_X_Sw_Ver_Tst_DWP)) >= 0) AND (USINT_TO_REAL(BYTE_TO_USINT(Raw_X_Sw_Ver_Tst_DWP)) <= 250));
GVL.IIVD.X_Sw_Ver_Tst_DWP.v					:= NOT( GVL.IIVD.S_TmOut_Arac_Bilgi_2_0X2E1 OR GVL.IIVD.X_Sw_Ver_Tst_DWP.RangeExcd OR GVL.IIVD.X_Sw_Ver_Tst_DWP.e OR GVL.IIVD.X_Sw_Ver_Tst_DWP.na) ;
GVL.IIVD.X_Sw_Ver_Tst_DWP.x					:= 
(*SELECT 1 : Is data valid ?*)					SEL(GVL.IIVD.X_Sw_Ver_Tst_DWP.v,
(*DEFAULT value assigment*)						0,
(*Transmission is VALID*)						USINT_TO_REAL(BYTE_TO_USINT(Raw_X_Sw_Ver_Tst_DWP)));	 
{endregion}	 
		  
{region " SIGNAL AREA : NAME->X_Sw_Ver_Mjr_VCU LENGTH->8 STARTBIT :24"}
Raw_X_Sw_Ver_Mjr_VCU						:= _FB_CanRx_Message_Unpack_2E1.X_Byte_3;
GVL.IIVD.X_Sw_Ver_Mjr_VCU.e					:= (Raw_X_Sw_Ver_Mjr_VCU > 16#FD) AND (Raw_X_Sw_Ver_Mjr_VCU < 16#FF);
GVL.IIVD.X_Sw_Ver_Mjr_VCU.na				:= (Raw_X_Sw_Ver_Mjr_VCU = 16#FF);
GVL.IIVD.X_Sw_Ver_Mjr_VCU.RangeExcd			:= NOT ((USINT_TO_REAL(BYTE_TO_USINT(Raw_X_Sw_Ver_Mjr_VCU)) >= 0) AND (USINT_TO_REAL(BYTE_TO_USINT(Raw_X_Sw_Ver_Mjr_VCU)) <= 250));
GVL.IIVD.X_Sw_Ver_Mjr_VCU.v					:= NOT( GVL.IIVD.S_TmOut_Arac_Bilgi_2_0X2E1 OR GVL.IIVD.X_Sw_Ver_Mjr_VCU.RangeExcd OR GVL.IIVD.X_Sw_Ver_Mjr_VCU.e OR GVL.IIVD.X_Sw_Ver_Mjr_VCU.na) ;
GVL.IIVD.X_Sw_Ver_Mjr_VCU.x					:= 
(*SELECT 1 : Is data valid ?*)					SEL(GVL.IIVD.X_Sw_Ver_Mjr_VCU.v,
(*DEFAULT value assigment*)						0,
(*Transmission is VALID*)						USINT_TO_REAL(BYTE_TO_USINT(Raw_X_Sw_Ver_Mjr_VCU)));	 
{endregion}	
		  
{region " SIGNAL AREA : NAME->X_Sw_Ver_Mnr_VCU LENGTH->8 STARTBIT :32"}
Raw_X_Sw_Ver_Mnr_VCU						:= _FB_CanRx_Message_Unpack_2E1.X_Byte_4;
GVL.IIVD.X_Sw_Ver_Mnr_VCU.e					:= (Raw_X_Sw_Ver_Mnr_VCU > 16#FD) AND (Raw_X_Sw_Ver_Mnr_VCU < 16#FF);
GVL.IIVD.X_Sw_Ver_Mnr_VCU.na				:= (Raw_X_Sw_Ver_Mnr_VCU = 16#FF);
GVL.IIVD.X_Sw_Ver_Mnr_VCU.RangeExcd			:= NOT ((USINT_TO_REAL(BYTE_TO_USINT(Raw_X_Sw_Ver_Mnr_VCU)) >= 0) AND (USINT_TO_REAL(BYTE_TO_USINT(Raw_X_Sw_Ver_Mnr_VCU)) <= 250));
GVL.IIVD.X_Sw_Ver_Mnr_VCU.v					:= NOT( GVL.IIVD.S_TmOut_Arac_Bilgi_2_0X2E1 OR GVL.IIVD.X_Sw_Ver_Mnr_VCU.RangeExcd OR GVL.IIVD.X_Sw_Ver_Mnr_VCU.e OR GVL.IIVD.X_Sw_Ver_Mnr_VCU.na) ;
GVL.IIVD.X_Sw_Ver_Mnr_VCU.x					:= 
(*SELECT 1 : Is data valid ?*)					SEL(GVL.IIVD.X_Sw_Ver_Mnr_VCU.v,
(*DEFAULT value assigment*)						0,
(*Transmission is VALID*)						USINT_TO_REAL(BYTE_TO_USINT(Raw_X_Sw_Ver_Mnr_VCU)));	 
{endregion}
		  
{region " SIGNAL AREA : NAME->X_Sw_Ver_Tst_VCU LENGTH->8 STARTBIT :40"}
Raw_X_Sw_Ver_Tst_VCU						:= _FB_CanRx_Message_Unpack_2E1.X_Byte_5;
GVL.IIVD.X_Sw_Ver_Tst_VCU.e					:= (Raw_X_Sw_Ver_Tst_VCU > 16#FD) AND (Raw_X_Sw_Ver_Tst_VCU < 16#FF);
GVL.IIVD.X_Sw_Ver_Tst_VCU.na				:= (Raw_X_Sw_Ver_Tst_VCU = 16#FF);
GVL.IIVD.X_Sw_Ver_Tst_VCU.RangeExcd			:= NOT ((USINT_TO_REAL(BYTE_TO_USINT(Raw_X_Sw_Ver_Tst_VCU)) >= 0) AND (USINT_TO_REAL(BYTE_TO_USINT(Raw_X_Sw_Ver_Tst_VCU)) <= 250));
GVL.IIVD.X_Sw_Ver_Tst_VCU.v					:= NOT( GVL.IIVD.S_TmOut_Arac_Bilgi_2_0X2E1 OR GVL.IIVD.X_Sw_Ver_Tst_VCU.RangeExcd OR GVL.IIVD.X_Sw_Ver_Tst_VCU.e OR GVL.IIVD.X_Sw_Ver_Tst_VCU.na) ;
GVL.IIVD.X_Sw_Ver_Tst_VCU.x					:= 
(*SELECT 1 : Is data valid ?*)					SEL(GVL.IIVD.X_Sw_Ver_Tst_VCU.v,
(*DEFAULT value assigment*)						0,
(*Transmission is VALID*)						USINT_TO_REAL(BYTE_TO_USINT(Raw_X_Sw_Ver_Tst_VCU)));	 
{endregion}		
		  
{region " SIGNAL AREA : NAME->X_Sw_Ver_Mjr_ATS LENGTH->8 STARTBIT :48"}
Raw_X_Sw_Ver_Mjr_ATS						:= _FB_CanRx_Message_Unpack_2E1.X_Byte_6;
GVL.IIVD.X_Sw_Ver_Mjr_ATS.e					:= (Raw_X_Sw_Ver_Mjr_ATS > 16#FD) AND (Raw_X_Sw_Ver_Mjr_ATS < 16#FF);
GVL.IIVD.X_Sw_Ver_Mjr_ATS.na				:= (Raw_X_Sw_Ver_Mjr_ATS = 16#FF);
GVL.IIVD.X_Sw_Ver_Mjr_ATS.RangeExcd			:= NOT ((USINT_TO_REAL(BYTE_TO_USINT(Raw_X_Sw_Ver_Mjr_ATS)) >= 0) AND (USINT_TO_REAL(BYTE_TO_USINT(Raw_X_Sw_Ver_Mjr_ATS)) <= 250));
GVL.IIVD.X_Sw_Ver_Mjr_ATS.v					:= NOT( GVL.IIVD.S_TmOut_Arac_Bilgi_2_0X2E1 OR GVL.IIVD.X_Sw_Ver_Mjr_ATS.RangeExcd OR GVL.IIVD.X_Sw_Ver_Mjr_ATS.e OR GVL.IIVD.X_Sw_Ver_Mjr_ATS.na) ;
GVL.IIVD.X_Sw_Ver_Mjr_ATS.x					:= 
(*SELECT 1 : Is data valid ?*)					SEL(GVL.IIVD.X_Sw_Ver_Mjr_ATS.v,
(*DEFAULT value assigment*)						0,
(*Transmission is VALID*)						USINT_TO_REAL(BYTE_TO_USINT(Raw_X_Sw_Ver_Mjr_ATS)));	 
{endregion}	
		  
{region " SIGNAL AREA : NAME->X_Sw_Ver_Mnr_ATS LENGTH->8 STARTBIT :54"}
Raw_X_Sw_Ver_Mnr_ATS						:= _FB_CanRx_Message_Unpack_2E1.X_Byte_7;
GVL.IIVD.X_Sw_Ver_Mnr_ATS.e					:= (Raw_X_Sw_Ver_Mnr_ATS > 16#FD) AND (Raw_X_Sw_Ver_Mnr_ATS < 16#FF);
GVL.IIVD.X_Sw_Ver_Mnr_ATS.na				:= (Raw_X_Sw_Ver_Mnr_ATS = 16#FF);
GVL.IIVD.X_Sw_Ver_Mnr_ATS.RangeExcd			:= NOT ((USINT_TO_REAL(BYTE_TO_USINT(Raw_X_Sw_Ver_Mnr_ATS)) >= 0) AND (USINT_TO_REAL(BYTE_TO_USINT(Raw_X_Sw_Ver_Mnr_ATS)) <= 250));
GVL.IIVD.X_Sw_Ver_Mnr_ATS.v					:= NOT( GVL.IIVD.S_TmOut_Arac_Bilgi_2_0X2E1 OR GVL.IIVD.X_Sw_Ver_Mnr_ATS.RangeExcd OR GVL.IIVD.X_Sw_Ver_Mnr_ATS.e OR GVL.IIVD.X_Sw_Ver_Mnr_ATS.na) ;
GVL.IIVD.X_Sw_Ver_Mnr_ATS.x					:= 
(*SELECT 1 : Is data valid ?*)					SEL(GVL.IIVD.X_Sw_Ver_Mnr_ATS.v,
(*DEFAULT value assigment*)						0,
(*Transmission is VALID*)						USINT_TO_REAL(BYTE_TO_USINT(Raw_X_Sw_Ver_Mnr_ATS)));	 
{endregion}	
{endregion}

{region " MESSAGE AREA :Diag_Temel_Durum- ID:300"}
_FB_CanRx_Message_Unpack_300 (		C_Enable	:= GVL.IIVD.S_CAN_Init,
     								Obj_CAN		:= ADR(GVL.IC.Obj_CAN0),
     								X_MsgID		:= 16#300,
     								Tm_MsgTmOut := TIME#500MS,
     								S_Extended	:= 0,
     								S_ER_TmOut	=> GVL.IIVD.S_TmOut_Diag_Temel_Durum_0X300);

{region " SIGNAL AREA : NAME->N_Diag_Lf LENGTH->8 STARTBIT :0"}
Raw_N_Diag_Lf								:= _FB_CanRx_Message_Unpack_300.X_Byte_0;
GVL.IIVD.N_Diag_Lf.e						:= (Raw_N_Diag_Lf > 16#FD) AND (Raw_N_Diag_Lf < 16#FF);
GVL.IIVD.N_Diag_Lf.na						:= (Raw_N_Diag_Lf = 16#FF);
GVL.IIVD.N_Diag_Lf.RangeExcd				:= NOT ((BYTE_TO_USINT(Raw_N_Diag_Lf) >= 0) AND (BYTE_TO_USINT(Raw_N_Diag_Lf) <= 250));
GVL.IIVD.N_Diag_Lf.v						:= NOT GVL.IIVD.S_TmOut_Diag_Temel_Durum_0X300 AND NOT GVL.IIVD.N_Diag_Lf.RangeExcd AND NOT GVL.IIVD.N_Diag_Lf.e AND NOT GVL.IIVD.N_Diag_Lf.na;
GVL.IIVD.N_Diag_Lf.x						:= 
(*SELECT 1 : Is data valid ?*)					SEL(GVL.IIVD.N_Diag_Lf.v,
(*DEFAULT value assigment*)						0,
(*Transmission is VALID*)						BYTE_TO_USINT(Raw_N_Diag_Lf));
{endregion}
// PR1006_SRS_000539_TIMTRO
{region " SIGNAL AREA : NAME->C_Set_Odo_Btn LENGTH->1 STARTBIT :9"}
GVL.IIVD.C_Set_Odo_Btn.v		:= NOT GVL.IIVD.S_TmOut_Diag_Temel_Durum_0X300;
GVL.IIVD.C_Set_Odo_Btn.x		:= GVL.IIVD.C_Set_Odo_Btn.v AND _FB_CanRx_Message_Unpack_300.S_Bit_9;
{endregion}
{region " SIGNAL AREA : NAME->S_Tst_Pg_Act LENGTH->2 STARTBIT :10"}
GVL.IIVD.S_Tst_Pg_Act.v						:= NOT GVL.IIVD.S_TmOut_Diag_Temel_Durum_0X300 AND NOT _FB_CanRx_Message_Unpack_300.S_Bit_11;
GVL.IIVD.S_Tst_Pg_Act.x						:= GVL.IIVD.S_Tst_Pg_Act.v AND _FB_CanRx_Message_Unpack_300.S_Bit_10;
GVL.IIVD.S_Tst_Pg_Act.e						:= _FB_CanRx_Message_Unpack_300.S_Bit_11 AND NOT _FB_CanRx_Message_Unpack_300.S_Bit_10 ;
GVL.IIVD.S_Tst_Pg_Act.na					:= _FB_CanRx_Message_Unpack_300.S_Bit_11 AND _FB_CanRx_Message_Unpack_300.S_Bit_10 ;
{endregion}
{region " SIGNAL AREA : NAME->S_Para_Pg_Act LENGTH->2 STARTBIT :12"}
GVL.IIVD.S_Para_Pg_Act.v					:= NOT GVL.IIVD.S_TmOut_Diag_Temel_Durum_0X300 AND NOT _FB_CanRx_Message_Unpack_300.S_Bit_13;
GVL.IIVD.S_Para_Pg_Act.x					:= GVL.IIVD.S_Para_Pg_Act.v AND _FB_CanRx_Message_Unpack_300.S_Bit_12;
GVL.IIVD.S_Para_Pg_Act.e					:= _FB_CanRx_Message_Unpack_300.S_Bit_13 AND NOT _FB_CanRx_Message_Unpack_300.S_Bit_12 ;
GVL.IIVD.S_Para_Pg_Act.na					:= _FB_CanRx_Message_Unpack_300.S_Bit_13 AND _FB_CanRx_Message_Unpack_300.S_Bit_12 ;
{endregion}
{region " SIGNAL AREA : NAME->S_HV_On_Btn LENGTH->1 STARTBIT :14"}
GVL.IIVD.S_HV_On_Btn.v						:= NOT GVL.IIVD.S_TmOut_Diag_Temel_Durum_0X300;
GVL.IIVD.S_HV_On_Btn.x						:= GVL.IIVD.S_HV_On_Btn.v AND _FB_CanRx_Message_Unpack_300.S_Bit_14;
{endregion}
{region " SIGNAL AREA : NAME->S_HV_Off_Btn LENGTH->1 STARTBIT :15"}
GVL.IIVD.S_HV_Off_Btn.v						:= NOT GVL.IIVD.S_TmOut_Diag_Temel_Durum_0X300;
GVL.IIVD.S_HV_Off_Btn.x						:= GVL.IIVD.S_HV_Off_Btn.v AND _FB_CanRx_Message_Unpack_300.S_Bit_15;
{endregion}
{region " SIGNAL AREA : NAME->S_Tm_Btn LENGTH->1 STARTBIT :16"}
GVL.IIVD.S_Tm_Btn.v							:= NOT GVL.IIVD.S_TmOut_Diag_Temel_Durum_0X300;
GVL.IIVD.S_Tm_Btn.x							:= GVL.IIVD.S_Tm_Btn.v AND _FB_CanRx_Message_Unpack_300.S_Bit_16;
{endregion}	
{region " SIGNAL AREA : NAME->S_Eep_Rst LENGTH->1 STARTBIT :17"}
GVL.IIVD.S_Eep_Rst.v						:= NOT GVL.IIVD.S_TmOut_Diag_Temel_Durum_0X300;
GVL.IIVD.S_Eep_Rst.x						:= GVL.IIVD.S_Eep_Rst.v AND _FB_CanRx_Message_Unpack_300.S_Bit_17;
{endregion}			
{region " SIGNAL AREA : NAME->C_Par_Rx LENGTH->1 STARTBIT :19"}
GVL.IIVD.C_Par_Rx.v							:= NOT GVL.IIVD.S_TmOut_Diag_Temel_Durum_0X300;
GVL.IIVD.C_Par_Rx.x							:= GVL.IIVD.C_Par_Rx.v AND _FB_CanRx_Message_Unpack_300.S_Bit_19;
{endregion}		  
{region " SIGNAL AREA : NAME->C_Par_Wr LENGTH->1 STARTBIT :20"}
GVL.IIVD.C_Par_Wr.v							:= NOT GVL.IIVD.S_TmOut_Diag_Temel_Durum_0X300;
GVL.IIVD.C_Par_Wr.x							:= GVL.IIVD.C_Par_Wr.v AND _FB_CanRx_Message_Unpack_300.S_Bit_20;
{endregion}	
{region " SIGNAL AREA : NAME->C_Clr_H LENGTH->1 STARTBIT :21"}
GVL.IIVD.C_Clr_EH.v							:= NOT GVL.IIVD.S_TmOut_Diag_Temel_Durum_0X300;
GVL.IIVD.C_Clr_EH.x							:= GVL.IIVD.C_Clr_EH.v AND _FB_CanRx_Message_Unpack_300.S_Bit_21;	 
{endregion}
// PR1006_SRS_000533_TIMTRO
{region " SIGNAL AREA : NAME->S_Sw_Ver_Incomp LENGTH->1 STARBIT:22"}
GVL.IIVD.S_Sw_Ver_Incomp.v					:= NOT GVL.IIVD.S_TmOut_Diag_Temel_Durum_0X300;
GVL.IIVD.S_Sw_Ver_Incomp.x					:= GVL.IIVD.S_Sw_Ver_Incomp.v AND _FB_CanRx_Message_Unpack_300.S_Bit_22;
{endregion}
{region " SIGNAL AREA : NAME->X_Minute LENGTH->8 STARTBIT :0"}
Raw_W_Rd_Par_ID								:= _FB_CanRx_Message_Unpack_300.X_Byte_3;
GVL.IIVD.W_Rd_Par_ID.e						:= (Raw_W_Rd_Par_ID > 16#FD) AND (Raw_W_Rd_Par_ID < 16#FF);
GVL.IIVD.W_Rd_Par_ID.na						:= (Raw_W_Rd_Par_ID = 16#FF);
GVL.IIVD.W_Rd_Par_ID.RangeExcd				:= NOT ((USINT_TO_REAL(BYTE_TO_USINT(Raw_W_Rd_Par_ID)) > 0) AND (USINT_TO_REAL(BYTE_TO_USINT(Raw_W_Rd_Par_ID)) <= 200));
GVL.IIVD.W_Rd_Par_ID.v						:= NOT( GVL.IIVD.S_TmOut_Diag_Temel_Durum_0X300 OR GVL.IIVD.W_Rd_Par_ID.RangeExcd OR GVL.IIVD.W_Rd_Par_ID.e OR GVL.IIVD.W_Rd_Par_ID.na) ;
GVL.IIVD.W_Rd_Par_ID.x						:= 
(*SELECT 1 : Is data valid ?*)					SEL(GVL.IIVD.W_Rd_Par_ID.v,
(*DEFAULT value assigment*)						1,
(*Transmission is VALID*)						USINT_TO_REAL(BYTE_TO_USINT(Raw_W_Rd_Par_ID)));
{endregion}			  
{region " SIGNAL AREA : NAME->W_Odo LENGTH->32 STARTBIT :32"}
_FB_PACK_BYTE_TO_DWORD_0 (	X_BYTE_0	:= _FB_CanRx_Message_Unpack_300.X_Byte_4, 
							X_BYTE_1	:= _FB_CanRx_Message_Unpack_300.X_Byte_5, 
							X_BYTE_2	:= _FB_CanRx_Message_Unpack_300.X_Byte_6, 
							X_BYTE_3	:= _FB_CanRx_Message_Unpack_300.X_Byte_7 , 
							X_DWORD_0 	=> Raw_W_Odo);
GVL.IIVD.W_Odo.e							:= (Raw_W_Odo > 16#FDFFFFFF) AND (Raw_W_Odo <= 16#FEFFFFFF);
GVL.IIVD.W_Odo.na							:= (Raw_W_Odo > 16#FEFFFFFF);
GVL.IIVD.W_Odo.RangeExcd					:= NOT ((UDINT_TO_REAL(DWORD_TO_UDINT(Raw_W_Odo))*0.1 >= 0) AND (UDINT_TO_REAL(DWORD_TO_UDINT(Raw_W_Odo))*0.1 <= 421108121.5));
GVL.IIVD.W_Odo.v							:= NOT( GVL.IIVD.S_TmOut_Diag_Temel_Durum_0X300 OR GVL.IIVD.W_Odo.RangeExcd OR GVL.IIVD.W_Odo.e OR GVL.IIVD.W_Odo.na) ;
GVL.IIVD.W_Odo.x							:= 
(*SELECT 1 : Is data valid ?*)					SEL(GVL.IIVD.W_Odo.v,
(*DEFAULT value assigment*)						0,
(*Transmission is VALID*)						UDINT_TO_REAL(DWORD_TO_UDINT(Raw_W_Odo))*0.1);
{endregion}
{endregion}

{region " MESSAGE AREA :Diag_RTC- ID:301"}

_FB_CanRx_Message_Unpack_301 (		C_Enable	:= GVL.IIVD.S_CAN_Init,
     								Obj_CAN		:= ADR(GVL.IC.Obj_CAN0),
     								X_MsgID		:= 16#301,
     								Tm_MsgTmOut	:= TIME#500MS,
     								S_Extended	:= 0,
     								S_ER_TmOut	=> GVL.IIVD.S_TmOut_Diag_RTC_0X301);

{region " SIGNAL AREA : NAME->X_Minute LENGTH->8 STARTBIT :0"}
Raw_X_Minute							:= _FB_CanRx_Message_Unpack_301.X_Byte_0;
GVL.IIVD.X_Minute.e						:= (Raw_X_Minute > 16#FD) AND (Raw_X_Minute < 16#FF);
GVL.IIVD.X_Minute.na					:= (Raw_X_Minute = 16#FF);
GVL.IIVD.X_Minute.RangeExcd				:= NOT ((USINT_TO_REAL(BYTE_TO_USINT(Raw_X_Minute)) >= 0) AND (USINT_TO_REAL(BYTE_TO_USINT(Raw_X_Minute)) <= 59));
GVL.IIVD.X_Minute.v						:= NOT( GVL.IIVD.S_TmOut_Diag_RTC_0X301 OR GVL.IIVD.X_Minute.RangeExcd OR GVL.IIVD.X_Minute.e OR GVL.IIVD.X_Minute.na) ;
GVL.IIVD.X_Minute.x						:= 
(*SELECT 1 : Is data valid ?*)				SEL(GVL.IIVD.X_Minute.v,
(*DEFAULT value assigment*)					0,
(*Transmission is VALID*)					USINT_TO_REAL(BYTE_TO_USINT(Raw_X_Minute)));
{endregion}
{region " SIGNAL AREA : NAME->X_Hour LENGTH->8 STARTBIT :8"}
Raw_X_Hour								:= _FB_CanRx_Message_Unpack_301.X_Byte_1;
GVL.IIVD.X_Hour.e						:= (Raw_X_Hour > 16#FD) AND (Raw_X_Hour < 16#FF);
GVL.IIVD.X_Hour.na						:= (Raw_X_Hour = 16#FF);
GVL.IIVD.X_Hour.RangeExcd				:= NOT ((USINT_TO_REAL(BYTE_TO_USINT(Raw_X_Hour)) >= 0) AND (USINT_TO_REAL(BYTE_TO_USINT(Raw_X_Hour)) <= 23));
GVL.IIVD.X_Hour.v						:= NOT( GVL.IIVD.S_TmOut_Diag_RTC_0X301 OR GVL.IIVD.X_Hour.RangeExcd OR GVL.IIVD.X_Hour.e OR GVL.IIVD.X_Hour.na) ;
GVL.IIVD.X_Hour.x						:= 
(*SELECT 1 : Is data valid ?*)				SEL(GVL.IIVD.X_Hour.v,
(*DEFAULT value assigment*)					0,
(*Transmission is VALID*)					USINT_TO_REAL(BYTE_TO_USINT(Raw_X_Hour)));
{endregion}
{region " SIGNAL AREA : NAME->X_Day LENGTH->8 STARTBIT :16"}
Raw_X_Day								:= _FB_CanRx_Message_Unpack_301.X_Byte_2;
GVL.IIVD.X_Day.e						:= (Raw_X_Day > 16#FD) AND (Raw_X_Day < 16#FF);
GVL.IIVD.X_Day.na						:= (Raw_X_Day = 16#FF);
GVL.IIVD.X_Day.RangeExcd				:= NOT ((USINT_TO_REAL(BYTE_TO_USINT(Raw_X_Day)) >= 0) AND (USINT_TO_REAL(BYTE_TO_USINT(Raw_X_Day)) <= 31));
GVL.IIVD.X_Day.v						:= NOT( GVL.IIVD.S_TmOut_Diag_RTC_0X301 OR GVL.IIVD.X_Day.RangeExcd OR GVL.IIVD.X_Day.e OR GVL.IIVD.X_Day.na) ;
GVL.IIVD.X_Day.x						:= 
(*SELECT 1 : Is data valid ?*)				SEL(GVL.IIVD.X_Day.v,
(*DEFAULT value assigment*)					0,
(*Transmission is VALID*)					USINT_TO_REAL(BYTE_TO_USINT(Raw_X_Day)));
{endregion}
{region " SIGNAL AREA : NAME->X_Month LENGTH->8 STARTBIT :24"}
Raw_X_Month								:= _FB_CanRx_Message_Unpack_301.X_Byte_3;
GVL.IIVD.X_Month.e						:= (Raw_X_Month > 16#FD) AND (Raw_X_Month < 16#FF);
GVL.IIVD.X_Month.na						:= (Raw_X_Month = 16#FF);
GVL.IIVD.X_Month.RangeExcd				:= NOT ((USINT_TO_REAL(BYTE_TO_USINT(Raw_X_Month)) >= 0) AND (USINT_TO_REAL(BYTE_TO_USINT(Raw_X_Month)) <= 12));
GVL.IIVD.X_Month.v						:= NOT( GVL.IIVD.S_TmOut_Diag_RTC_0X301 OR GVL.IIVD.X_Month.RangeExcd OR GVL.IIVD.X_Month.e OR GVL.IIVD.X_Month.na) ;
GVL.IIVD.X_Month.x						:= 
(*SELECT 1 : Is data valid ?*)				SEL(GVL.IIVD.X_Month.v,
(*DEFAULT value assigment*)					0,
(*Transmission is VALID*)					USINT_TO_REAL(BYTE_TO_USINT(Raw_X_Month)));
{endregion}
{region " SIGNAL AREA : NAME->X_Year LENGTH->8 STARTBIT :32"}
Raw_X_Year								:= _FB_CanRx_Message_Unpack_301.X_Byte_4;
GVL.IIVD.X_Year.e						:= (Raw_X_Year > 16#FD) AND (Raw_X_Year < 16#FF);
GVL.IIVD.X_Year.na						:= (Raw_X_Year = 16#FF);
GVL.IIVD.X_Year.RangeExcd				:= NOT ((USINT_TO_REAL(BYTE_TO_USINT(Raw_X_Year))+(1985) >= 1985) AND (USINT_TO_REAL(BYTE_TO_USINT(Raw_X_Year))+(1985) <= 2230));
GVL.IIVD.X_Year.v						:= NOT( GVL.IIVD.S_TmOut_Diag_RTC_0X301 OR GVL.IIVD.X_Year.RangeExcd OR GVL.IIVD.X_Year.e OR GVL.IIVD.X_Year.na) ;
GVL.IIVD.X_Year.x						:= 
(*SELECT 1 : Is data valid ?*)				SEL(GVL.IIVD.X_Year.v,
(*DEFAULT value assigment*)					1985,
(*Transmission is VALID*)					USINT_TO_REAL(BYTE_TO_USINT(Raw_X_Year))+(1985));
{endregion}
{endregion}


{region " MESSAGE AREA :Diag_Parameter- ID:302"}

_FB_CanRx_Message_Unpack_302 (		C_Enable	:= GVL.IIVD.S_CAN_Init,
     								Obj_CAN		:= ADR(GVL.IC.Obj_CAN0),
     								X_MsgID		:= 16#302,
     								Tm_MsgTmOut	:= TIME#500MS,
     								S_Extended	:= 0,
     								S_ER_TmOut	=> GVL.IIVD.S_TmOut_Diag_Parameter_0X302);

GVL.IIVD.X_Param_Arr.X_No				:= SEL(_FB_CanRx_Message_Unpack_302.X_Byte_0 <> 0, 1,_FB_CanRx_Message_Unpack_302.X_Byte_0);	
GVL.IIVD.X_Param_Arr.X_Usr_Id			:= _FB_CanRx_Message_Unpack_302.X_Byte_1;	

_FB_PACK_BYTE_TO_WORD_5 (	X_BYTE_0	:= _FB_CanRx_Message_Unpack_302.X_Byte_2, 
							X_BYTE_1	:= _FB_CanRx_Message_Unpack_302.X_Byte_3, 
							X_WORD_0 	=> Raw_X_Par_Val);
GVL.IIVD.X_Param_Arr.X_Val				:= Raw_X_Par_Val;
GVL.IIVD.X_Param_Arr.X_Days				:= _FB_CanRx_Message_Unpack_302.X_Byte_4;								 
		  
_FB_PACK_8BITS_TO_BYTE_5 (	S_BIT_0		:= _FB_CanRx_Message_Unpack_302.S_Bit_40,
							S_BIT_1		:= _FB_CanRx_Message_Unpack_302.S_Bit_41,
							S_BIT_2		:= _FB_CanRx_Message_Unpack_302.S_Bit_42,
							S_BIT_3		:= _FB_CanRx_Message_Unpack_302.S_Bit_43,
							S_BIT_4		:= 0,
							S_BIT_5		:= 0,
							S_BIT_6		:= 0,
							S_BIT_7		:= 0,
							X_BYTE_0	=> Raw_X_Par_Month);
GVL.IIVD.X_Param_Arr.X_Months			:= Raw_X_Par_Month;								

_FB_PACK_8BITS_TO_BYTE_6 (	S_BIT_0		:= _FB_CanRx_Message_Unpack_302.S_Bit_44,
							S_BIT_1		:= _FB_CanRx_Message_Unpack_302.S_Bit_45,
							S_BIT_2		:= _FB_CanRx_Message_Unpack_302.S_Bit_46,
							S_BIT_3		:= _FB_CanRx_Message_Unpack_302.S_Bit_47,
							S_BIT_4		:= 0,
							S_BIT_5		:= 0,
							S_BIT_6		:= 0,
							S_BIT_7		:= 0,
							X_BYTE_0	=>Raw_X_Par_Year);
GVL.IIVD.X_Param_Arr.X_Years			:= Raw_X_Par_Year;			
GVL.IIVD.X_Param_Arr.X_Hours			:= _FB_CanRx_Message_Unpack_302.X_Byte_6;
GVL.IIVD.X_Param_Arr.X_Minutes			:= _FB_CanRx_Message_Unpack_302.X_Byte_7;	   		
{endregion}

{region " MESSAGE AREA :Diag_Op_Rst- ID:303"}
_FB_CanRx_Message_Unpack_303	(	C_Enable	:= GVL.IIVD.S_CAN_Init, 
									Obj_CAN		:= ADR(GVL.IC.Obj_CAN0), 
									X_MsgID		:= 16#303, 
									Tm_MsgTmOut	:= TIME#500MS, 
									S_Extended	:= 0, 
									S_ER_TmOut	=> GVL.IIVD.S_TmOut_Diag_Op_Rst_0X303);

{region " SIGNAL AREA : NAME->C_Rst_Tm_HVAC_On LENGTH->1 STARTBIT:0"}
GVL.IIVD.C_Rst_Tm_HVAC_On.v				:= NOT GVL.IIVD.S_TmOut_Diag_Op_Rst_0X303;
GVL.IIVD.C_Rst_Tm_HVAC_On.x				:= GVL.IIVD.C_Rst_Tm_HVAC_On.v AND _FB_CanRx_Message_Unpack_303.S_Bit_0;
{endregion}

{region " SIGNAL AREA : NAME->C_Rst_Drv_Op_Cnt LENGTH->1 STARTBIT:1"}
GVL.IIVD.C_Rst_Drv_Op_Cnt.v				:= NOT GVL.IIVD.S_TmOut_Diag_Op_Rst_0X303;
GVL.IIVD.C_Rst_Drv_Op_Cnt.x				:= GVL.IIVD.C_Rst_Drv_Op_Cnt.v AND _FB_CanRx_Message_Unpack_303.S_Bit_1;
{endregion}

{region " SIGNAL AREA : NAME->C_Rst_Pass1_Op_Cnt LENGTH->1 STARTBIT:2"}
GVL.IIVD.C_Rst_Pass1_Op_Cnt.v			:= NOT GVL.IIVD.S_TmOut_Diag_Op_Rst_0X303;
GVL.IIVD.C_Rst_Pass1_Op_Cnt.x			:= GVL.IIVD.C_Rst_Pass1_Op_Cnt.v AND _FB_CanRx_Message_Unpack_303.S_Bit_2;
{endregion}

{region " SIGNAL AREA : NAME->C_Rst_Pass2_Op_Cnt LENGTH->1 STARTBIT:3"}
GVL.IIVD.C_Rst_Pass2_Op_Cnt.v			:= NOT GVL.IIVD.S_TmOut_Diag_Op_Rst_0X303;
GVL.IIVD.C_Rst_Pass2_Op_Cnt.x			:= GVL.IIVD.C_Rst_Pass2_Op_Cnt.v AND _FB_CanRx_Message_Unpack_303.S_Bit_3;
{endregion}

{region " SIGNAL AREA : NAME->C_Rst_Dr1_Cycle LENGTH->1 STARTBIT:4"}
GVL.IIVD.C_Rst_Dr1_Cycle.v				:= NOT GVL.IIVD.S_TmOut_Diag_Op_Rst_0X303;
GVL.IIVD.C_Rst_Dr1_Cycle.x				:= GVL.IIVD.C_Rst_Dr1_Cycle.v AND _FB_CanRx_Message_Unpack_303.S_Bit_4;
{endregion}

{region " SIGNAL AREA : NAME->C_Rst_Dr2_Cycle LENGTH->1 STARTBIT:5"}
GVL.IIVD.C_Rst_Dr2_Cycle.v				:= NOT GVL.IIVD.S_TmOut_Diag_Op_Rst_0X303;
GVL.IIVD.C_Rst_Dr2_Cycle.x				:= GVL.IIVD.C_Rst_Dr2_Cycle.v AND _FB_CanRx_Message_Unpack_303.S_Bit_5;
{endregion}

{region " SIGNAL AREA : NAME->C_Rst_Dr3_Cycle LENGTH->1 STARTBIT:6"}
GVL.IIVD.C_Rst_Dr3_Cycle.v				:= NOT GVL.IIVD.S_TmOut_Diag_Op_Rst_0X303;
GVL.IIVD.C_Rst_Dr3_Cycle.x				:= GVL.IIVD.C_Rst_Dr3_Cycle.v AND _FB_CanRx_Message_Unpack_303.S_Bit_6;
{endregion}

{region " SIGNAL AREA : NAME->C_Rst_Dr4_Cycle LENGTH->1 STARTBIT:7"}
GVL.IIVD.C_Rst_Dr4_Cycle.v				:= NOT GVL.IIVD.S_TmOut_Diag_Op_Rst_0X303;
GVL.IIVD.C_Rst_Dr4_Cycle.x				:= GVL.IIVD.C_Rst_Drv_Op_Cnt.v AND _FB_CanRx_Message_Unpack_303.S_Bit_7;
{endregion}
{endregion} 

{region " MESSAGE AREA :ECU_Dijital_Cikis_Test- ID:310"}

_FB_CanRx_Message_Unpack_310 (		C_Enable:= GVL.IIVD.S_CAN_Init,
     								Obj_CAN:= ADR(GVL.IC.Obj_CAN0),
     								X_MsgID:= 16#310,
     								Tm_MsgTmOut:= TIME#500ms,
     								S_Extended:= 0,
     								S_ER_TmOut=> GVL.IIVD.S_TmOut_ECU_Dijital_Cikis_Test_0X310);

{region " SIGNAL AREA : NAME->S_Tst_HV_On LENGTH->1 STARTBIT :34"}
GVL.IIVD.S_Tst_HV_On.v					:= NOT GVL.IIVD.S_TmOut_ECU_Dijital_Cikis_Test_0X310;
GVL.IIVD.S_Tst_HV_On.x					:= GVL.IIVD.S_Tst_HV_On.v AND _FB_CanRx_Message_Unpack_310.S_Bit_34;
{endregion}
{region " SIGNAL AREA : NAME->S_Tst_TCU_CAN_Sp LENGTH->1 STARTBIT :37"}
GVL.IIVD.S_Tst_TCU_CAN_Sp.v				:= NOT GVL.IIVD.S_TmOut_ECU_Dijital_Cikis_Test_0X310;
GVL.IIVD.S_Tst_TCU_CAN_Sp.x				:= GVL.IIVD.S_Tst_TCU_CAN_Sp.v AND _FB_CanRx_Message_Unpack_310.S_Bit_37;
{endregion}
{region " SIGNAL AREA : NAME->S_Tst_TCU_HV_On LENGTH->1 STARTBIT :38"}
GVL.IIVD.S_Tst_TCU_HV_On.v				:= NOT GVL.IIVD.S_TmOut_ECU_Dijital_Cikis_Test_0X310;
GVL.IIVD.S_Tst_TCU_HV_On.x				:= GVL.IIVD.S_Tst_TCU_HV_On.v AND _FB_CanRx_Message_Unpack_310.S_Bit_38;
{endregion}
{region " SIGNAL AREA : NAME->S_Tst_Air_Cmp_On LENGTH->1 STARTBIT :39"}
GVL.IIVD.S_Tst_Air_Cmp_On.v				:= NOT GVL.IIVD.S_TmOut_ECU_Dijital_Cikis_Test_0X310;
GVL.IIVD.S_Tst_Air_Cmp_On.x				:= GVL.IIVD.S_Tst_Air_Cmp_On.v AND _FB_CanRx_Message_Unpack_310.S_Bit_39;
{endregion}
{region " SIGNAL AREA : NAME->S_BMS_Wkup_Btn LENGTH->1 STARTBIT :40"}
GVL.IIVD.S_BMS_Wkup_Btn.v				:= NOT GVL.IIVD.S_TmOut_ECU_Dijital_Cikis_Test_0X310;
GVL.IIVD.S_BMS_Wkup_Btn.x				:= GVL.IIVD.S_BMS_Wkup_Btn.v AND _FB_CanRx_Message_Unpack_310.S_Bit_40;
{endregion}
{region " SIGNAL AREA : NAME->S_Mot_Fan_Ct_Btn LENGTH->1 STARTBIT :41"}
GVL.IIVD.S_Mot_Fan_Ct_Btn.v				:= NOT GVL.IIVD.S_TmOut_ECU_Dijital_Cikis_Test_0X310;
GVL.IIVD.S_Mot_Fan_Ct_Btn.x				:= GVL.IIVD.S_Mot_Fan_Ct_Btn.v AND _FB_CanRx_Message_Unpack_310.S_Bit_41;
{endregion}
{endregion}
 
{region " MESSAGE AREA :test sürüsü - ID:500"}

_FB_CanRx_Message_500 (		C_Enable	:= GVL.IIVD.S_CAN_Init,
     						Obj_CAN		:= ADR(GVL.IC.Obj_CAN0),
     						X_MsgID		:= 16#500,
     						Tm_MsgTmOut	:= TIME#2500MS,
     						S_Extended	:= 0,
     						S_ER_TmOut	=> );

{region " SIGNAL AREA : NAME->X_Axl1_Brk_Ling_1 LENGTH->8 STARTBIT :0"}
Raw_X_Spd_Max							:= _FB_CanRx_Message_500.X_Byte_0;
GVL.IIVD.X_Spd_Max.e					:= (Raw_X_Spd_Max > 16#FD) AND (Raw_X_Spd_Max < 16#FF);
GVL.IIVD.X_Spd_Max.na					:= (Raw_X_Spd_Max = 16#FF);
GVL.IIVD.X_Spd_Max.RangeExcd			:= NOT ((USINT_TO_REAL(BYTE_TO_USINT(Raw_X_Spd_Max)) >= 0) AND (USINT_TO_REAL(BYTE_TO_USINT(Raw_X_Spd_Max)) <= 100));
GVL.IIVD.X_Spd_Max.v					:= NOT( _FB_CanRx_Message_500.S_ER_TmOut OR GVL.IIVD.X_Spd_Max.RangeExcd OR GVL.IIVD.X_Spd_Max.e OR GVL.IIVD.X_Spd_Max.na) ;
GVL.IIVD.X_Spd_Max.x					:= 
(*SELECT 1 : Is data valid ?*)				SEL(GVL.IIVD.X_Spd_Max.v,
(*DEFAULT value assigment*)					80,
(*Transmission is VALID*)					USINT_TO_REAL(BYTE_TO_USINT(Raw_X_Spd_Max)));
{endregion}	 	 
{endregion}	
 
{region " MESSAGE AREA :Basamak Isitici Durumlari - ID:412"}

_FB_CanRx_Message_Unpack_412 (	C_Enable	:= GVL.IIVD.S_CAN_Init, 
								Obj_CAN		:= ADR(GVL.IC.Obj_CAN0), 
								X_MsgID		:= 16#412, 
								Tm_MsgTmOut	:= TIME#5000MS, 
								S_Extended	:= FALSE, 				// PR1006_REV_002374_TIMTRO
								S_ER_TmOut	=> GVL.IIVD.S_TmOut_Basamak_Isitici_Durumlari_0X412);

{region " SIGNAL AREA : NAME->C_Flr_Heat_1_Ct LENGTH->1 STARTBIT :0"}
GVL.IIVD.C_Flr_Heat_1_Ct.v			:= NOT GVL.IIVD.S_TmOut_Basamak_Isitici_Durumlari_0X412;
GVL.IIVD.C_Flr_Heat_1_Ct.x			:= GVL.IIVD.C_Flr_Heat_1_Ct.v AND _FB_CanRx_Message_Unpack_412.S_Bit_0;
{endregion}

{region " SIGNAL AREA : NAME->C_Flr_Heat_2_Ct LENGTH->1 STARTBIT :1"}
GVL.IIVD.C_Flr_Heat_2_Ct.v			:= NOT GVL.IIVD.S_TmOut_Basamak_Isitici_Durumlari_0X412;
GVL.IIVD.C_Flr_Heat_2_Ct.x			:= GVL.IIVD.C_Flr_Heat_2_Ct.v AND _FB_CanRx_Message_Unpack_412.S_Bit_1;
{endregion}

{region " SIGNAL AREA : NAME->C_Flr_Heat_3_Ct LENGTH->1 STARTBIT :2"}
GVL.IIVD.C_Flr_Heat_3_Ct.v			:= NOT GVL.IIVD.S_TmOut_Basamak_Isitici_Durumlari_0X412;
GVL.IIVD.C_Flr_Heat_3_Ct.x			:= GVL.IIVD.C_Flr_Heat_3_Ct.v AND _FB_CanRx_Message_Unpack_412.S_Bit_2;
{endregion}

{region " SIGNAL AREA : NAME->C_Flr_Heat_4_Ct LENGTH->1 STARTBIT :3"}
GVL.IIVD.C_Flr_Heat_4_Ct.v			:= NOT GVL.IIVD.S_TmOut_Basamak_Isitici_Durumlari_0X412;
GVL.IIVD.C_Flr_Heat_4_Ct.x			:= GVL.IIVD.C_Flr_Heat_4_Ct.v AND _FB_CanRx_Message_Unpack_412.S_Bit_3;
{endregion}

{region " SIGNAL AREA : NAME->C_Flr_Heat_5_Ct LENGTH->1 STARTBIT :4"}
GVL.IIVD.C_Flr_Heat_5_Ct.v			:= NOT GVL.IIVD.S_TmOut_Basamak_Isitici_Durumlari_0X412;
GVL.IIVD.C_Flr_Heat_5_Ct.x			:= GVL.IIVD.C_Flr_Heat_5_Ct.v AND _FB_CanRx_Message_Unpack_412.S_Bit_4;
{endregion}

{region " SIGNAL AREA : NAME->C_Flr_Heat_6_Ct LENGTH->1 STARTBIT :5"}
GVL.IIVD.C_Flr_Heat_6_Ct.v			:= NOT GVL.IIVD.S_TmOut_Basamak_Isitici_Durumlari_0X412;
GVL.IIVD.C_Flr_Heat_6_Ct.x			:= GVL.IIVD.C_Flr_Heat_6_Ct.v AND _FB_CanRx_Message_Unpack_412.S_Bit_5;
{endregion}

{region " SIGNAL AREA : NAME->S_Flr_Heat_1 LENGTH->1 STARTBIT :8"}
GVL.IIVD.S_Flr_Heat_1.v				:= NOT GVL.IIVD.S_TmOut_Basamak_Isitici_Durumlari_0X412;
GVL.IIVD.S_Flr_Heat_1.x				:= GVL.IIVD.S_Flr_Heat_1.v AND _FB_CanRx_Message_Unpack_412.S_Bit_8;
{endregion}

{region " SIGNAL AREA : NAME->S_Flr_Heat_2 LENGTH->1 STARTBIT :9"}
GVL.IIVD.S_Flr_Heat_2.v				:= NOT GVL.IIVD.S_TmOut_Basamak_Isitici_Durumlari_0X412;
GVL.IIVD.S_Flr_Heat_2.x				:= GVL.IIVD.S_Flr_Heat_2.v AND _FB_CanRx_Message_Unpack_412.S_Bit_9;
{endregion}

{region " SIGNAL AREA : NAME->S_Flr_Heat_3 LENGTH->1 STARTBIT :10"}
GVL.IIVD.S_Flr_Heat_3.v				:= NOT GVL.IIVD.S_TmOut_Basamak_Isitici_Durumlari_0X412;
GVL.IIVD.S_Flr_Heat_3.x				:= GVL.IIVD.S_Flr_Heat_3.v AND _FB_CanRx_Message_Unpack_412.S_Bit_10;
{endregion}

{region " SIGNAL AREA : NAME->S_Flr_Heat_4 LENGTH->1 STARTBIT :11"}
GVL.IIVD.S_Flr_Heat_4.v				:= NOT GVL.IIVD.S_TmOut_Basamak_Isitici_Durumlari_0X412;
GVL.IIVD.S_Flr_Heat_4.x				:= GVL.IIVD.S_Flr_Heat_4.v AND _FB_CanRx_Message_Unpack_412.S_Bit_11;
{endregion}

{region " SIGNAL AREA : NAME->S_Flr_Heat_5 LENGTH->1 STARTBIT :12"}
GVL.IIVD.S_Flr_Heat_5.v				:= NOT GVL.IIVD.S_TmOut_Basamak_Isitici_Durumlari_0X412;
GVL.IIVD.S_Flr_Heat_5.x				:= GVL.IIVD.S_Flr_Heat_5.v AND _FB_CanRx_Message_Unpack_412.S_Bit_12;
{endregion}

{region " SIGNAL AREA : NAME->S_Flr_Heat_6 LENGTH->1 STARTBIT :13"}
GVL.IIVD.S_Flr_Heat_6.v				:= NOT GVL.IIVD.S_TmOut_Basamak_Isitici_Durumlari_0X412;
GVL.IIVD.S_Flr_Heat_6.x				:= GVL.IIVD.S_Flr_Heat_6.v AND _FB_CanRx_Message_Unpack_412.S_Bit_13;
{endregion}

{region " SIGNAL AREA : NAME->S_Flr_Heat_1_Fan_Actv LENGTH->1 STARTBIT :16"}
GVL.IIVD.S_Flr_Heat_1_Fan_Actv.v	:= NOT GVL.IIVD.S_TmOut_Basamak_Isitici_Durumlari_0X412;
GVL.IIVD.S_Flr_Heat_1_Fan_Actv.x	:= GVL.IIVD.S_Flr_Heat_1_Fan_Actv.v AND _FB_CanRx_Message_Unpack_412.S_Bit_16;
{endregion}

{region " SIGNAL AREA : NAME->S_Flr_Heat_2_Fan_Actv LENGTH->1 STARTBIT :17"}
GVL.IIVD.S_Flr_Heat_2_Fan_Actv.v	:= NOT GVL.IIVD.S_TmOut_Basamak_Isitici_Durumlari_0X412;
GVL.IIVD.S_Flr_Heat_2_Fan_Actv.x	:= GVL.IIVD.S_Flr_Heat_2_Fan_Actv.v AND _FB_CanRx_Message_Unpack_412.S_Bit_17;
{endregion}

{region " SIGNAL AREA : NAME->S_Flr_Heat_3_Fan_Actv LENGTH->1 STARTBIT :18"}
GVL.IIVD.S_Flr_Heat_3_Fan_Actv.v	:= NOT GVL.IIVD.S_TmOut_Basamak_Isitici_Durumlari_0X412;
GVL.IIVD.S_Flr_Heat_3_Fan_Actv.x	:= GVL.IIVD.S_Flr_Heat_2_Fan_Actv.v AND _FB_CanRx_Message_Unpack_412.S_Bit_18;
{endregion}

{region " SIGNAL AREA : NAME->S_Flr_Heat_4_Fan_Actv LENGTH->1 STARTBIT :19"}
GVL.IIVD.S_Flr_Heat_4_Fan_Actv.v	:= NOT GVL.IIVD.S_TmOut_Basamak_Isitici_Durumlari_0X412;
GVL.IIVD.S_Flr_Heat_4_Fan_Actv.x	:= GVL.IIVD.S_Flr_Heat_4_Fan_Actv.v AND _FB_CanRx_Message_Unpack_412.S_Bit_19;
{endregion}

{region " SIGNAL AREA : NAME->S_Flr_Heat_5_Fan_Actv LENGTH->1 STARTBIT :20"}
GVL.IIVD.S_Flr_Heat_5_Fan_Actv.v	:= NOT GVL.IIVD.S_TmOut_Basamak_Isitici_Durumlari_0X412;
GVL.IIVD.S_Flr_Heat_5_Fan_Actv.x	:= GVL.IIVD.S_Flr_Heat_5_Fan_Actv.v AND _FB_CanRx_Message_Unpack_412.S_Bit_20;
{endregion}

{region " SIGNAL AREA : NAME->S_Flr_Heat_6_Fan_Actv LENGTH->1 STARTBIT :21"}
GVL.IIVD.S_Flr_Heat_6_Fan_Actv.v	:= NOT GVL.IIVD.S_TmOut_Basamak_Isitici_Durumlari_0X412;
GVL.IIVD.S_Flr_Heat_6_Fan_Actv.x	:= GVL.IIVD.S_Flr_Heat_6_Fan_Actv.v AND _FB_CanRx_Message_Unpack_412.S_Bit_21;
{endregion}

{region " SIGNAL AREA : NAME->S_Flr_Heat_1_Fus_Blw LENGTH->1 STARTBIT :24"}
GVL.IIVD.S_Flr_Heat_1_Fus_Blw.v		:= NOT GVL.IIVD.S_TmOut_Basamak_Isitici_Durumlari_0X412;
GVL.IIVD.S_Flr_Heat_1_Fus_Blw.x		:= GVL.IIVD.S_Flr_Heat_1_Fus_Blw.v AND _FB_CanRx_Message_Unpack_412.S_Bit_24;
{endregion}

{region " SIGNAL AREA : NAME->S_Flr_Heat_2_Fus_Blw LENGTH->1 STARTBIT :25"}
GVL.IIVD.S_Flr_Heat_2_Fus_Blw.v		:= NOT GVL.IIVD.S_TmOut_Basamak_Isitici_Durumlari_0X412;
GVL.IIVD.S_Flr_Heat_2_Fus_Blw.x		:= GVL.IIVD.S_Flr_Heat_2_Fus_Blw.v AND _FB_CanRx_Message_Unpack_412.S_Bit_25;
{endregion}

{region " SIGNAL AREA : NAME->S_Flr_Heat_3_Fus_Blw LENGTH->1 STARTBIT :26"}
GVL.IIVD.S_Flr_Heat_3_Fus_Blw.v		:= NOT GVL.IIVD.S_TmOut_Basamak_Isitici_Durumlari_0X412;
GVL.IIVD.S_Flr_Heat_3_Fus_Blw.x		:= GVL.IIVD.S_Flr_Heat_3_Fus_Blw.v AND _FB_CanRx_Message_Unpack_412.S_Bit_26;
{endregion}

{region " SIGNAL AREA : NAME->S_Flr_Heat_4_Fus_Blw LENGTH->1 STARTBIT :27"}
GVL.IIVD.S_Flr_Heat_4_Fus_Blw.v		:= NOT GVL.IIVD.S_TmOut_Basamak_Isitici_Durumlari_0X412;
GVL.IIVD.S_Flr_Heat_4_Fus_Blw.x		:= GVL.IIVD.S_Flr_Heat_4_Fus_Blw.v AND _FB_CanRx_Message_Unpack_412.S_Bit_27;
{endregion}

{region " SIGNAL AREA : NAME->S_Flr_Heat_5_Fus_Blw LENGTH->1 STARTBIT :28"}
GVL.IIVD.S_Flr_Heat_5_Fus_Blw.v		:= NOT GVL.IIVD.S_TmOut_Basamak_Isitici_Durumlari_0X412;
GVL.IIVD.S_Flr_Heat_5_Fus_Blw.x		:= GVL.IIVD.S_Flr_Heat_5_Fus_Blw.v AND _FB_CanRx_Message_Unpack_412.S_Bit_28;
{endregion}

{region " SIGNAL AREA : NAME->S_Flr_Heat_6_Fus_Blw LENGTH->1 STARTBIT :29"}
GVL.IIVD.S_Flr_Heat_6_Fus_Blw.v		:= NOT GVL.IIVD.S_TmOut_Basamak_Isitici_Durumlari_0X412;
GVL.IIVD.S_Flr_Heat_6_Fus_Blw.x		:= GVL.IIVD.S_Flr_Heat_6_Fus_Blw.v AND _FB_CanRx_Message_Unpack_412.S_Bit_29;
{endregion}

{region " SIGNAL AREA : NAME->S_ER_Flr_Heat_1_Thstat LENGTH->1 STARTBIT :32"}
GVL.IIVD.S_ER_Flr_Heat_1_Thstat.v	:= NOT GVL.IIVD.S_TmOut_Basamak_Isitici_Durumlari_0X412;
GVL.IIVD.S_ER_Flr_Heat_1_Thstat.x	:= GVL.IIVD.S_ER_Flr_Heat_1_Thstat.v AND _FB_CanRx_Message_Unpack_412.S_Bit_32;
{endregion}

{region " SIGNAL AREA : NAME->S_ER_Flr_Heat_2_Thstat LENGTH->1 STARTBIT :33"}
GVL.IIVD.S_ER_Flr_Heat_2_Thstat.v	:= NOT GVL.IIVD.S_TmOut_Basamak_Isitici_Durumlari_0X412;
GVL.IIVD.S_ER_Flr_Heat_2_Thstat.x	:= GVL.IIVD.S_ER_Flr_Heat_2_Thstat.v AND _FB_CanRx_Message_Unpack_412.S_Bit_33;
{endregion}

{region " SIGNAL AREA : NAME->S_ER_Flr_Heat_3_Thstat LENGTH->1 STARTBIT :34"}
GVL.IIVD.S_ER_Flr_Heat_3_Thstat.v	:= NOT GVL.IIVD.S_TmOut_Basamak_Isitici_Durumlari_0X412;
GVL.IIVD.S_ER_Flr_Heat_3_Thstat.x	:= GVL.IIVD.S_ER_Flr_Heat_3_Thstat.v AND _FB_CanRx_Message_Unpack_412.S_Bit_34;
{endregion}

{region " SIGNAL AREA : NAME->S_ER_Flr_Heat_4_Thstat LENGTH->1 STARTBIT :35"}
GVL.IIVD.S_ER_Flr_Heat_4_Thstat.v	:= NOT GVL.IIVD.S_TmOut_Basamak_Isitici_Durumlari_0X412;
GVL.IIVD.S_ER_Flr_Heat_4_Thstat.x	:= GVL.IIVD.S_ER_Flr_Heat_4_Thstat.v AND _FB_CanRx_Message_Unpack_412.S_Bit_35;
{endregion}

{region " SIGNAL AREA : NAME->S_ER_Flr_Heat_5_Thstat LENGTH->1 STARTBIT :36"}
GVL.IIVD.S_ER_Flr_Heat_5_Thstat.v	:= NOT GVL.IIVD.S_TmOut_Basamak_Isitici_Durumlari_0X412;
GVL.IIVD.S_ER_Flr_Heat_5_Thstat.x	:= GVL.IIVD.S_ER_Flr_Heat_5_Thstat.v AND _FB_CanRx_Message_Unpack_412.S_Bit_36;
{endregion}

{region " SIGNAL AREA : NAME->S_ER_Flr_Heat_6_Thstat LENGTH->1 STARTBIT :37"}
GVL.IIVD.S_ER_Flr_Heat_6_Thstat.v	:= NOT GVL.IIVD.S_TmOut_Basamak_Isitici_Durumlari_0X412;
GVL.IIVD.S_ER_Flr_Heat_6_Thstat.x	:= GVL.IIVD.S_ER_Flr_Heat_6_Thstat.v AND _FB_CanRx_Message_Unpack_412.S_Bit_37;
{endregion}

{region " SIGNAL AREA : NAME->X_T_Flr_1 LENGTH->8 STARTBIT :40"}
Raw_X_T_Flr_1						:= _FB_CanRx_Message_Unpack_412.X_Byte_5;
GVL.IIVD.X_T_Flr_1.e				:= (Raw_X_T_Flr_1 > 16#FD) AND (Raw_X_T_Flr_1 < 16#FF);
GVL.IIVD.X_T_Flr_1.na				:= (Raw_X_T_Flr_1 = 16#FF);
GVL.IIVD.X_T_Flr_1.RangeExcd		:= NOT ((USINT_TO_REAL(BYTE_TO_USINT(Raw_X_T_Flr_1)) >= -40) AND (USINT_TO_REAL(BYTE_TO_USINT(Raw_X_T_Flr_1)) <= 100));
GVL.IIVD.X_T_Flr_1.v				:= NOT (_FB_CanRx_Message_Unpack_412.S_ER_TmOut OR GVL.IIVD.X_T_Flr_1.RangeExcd OR GVL.IIVD.X_T_Flr_1.e OR GVL.IIVD.X_T_Flr_1.na) ;
GVL.IIVD.X_T_Flr_1.x				:= 
(*SELECT 1 : Is data valid ?*)			SEL(GVL.IIVD.X_T_Flr_1.v,
(*DEFAULT value assigment*)				0,
(*Transmission is VALID*)				USINT_TO_REAL(BYTE_TO_USINT(Raw_X_T_Flr_1)) );
{endregion}

{region " SIGNAL AREA : NAME->X_T_Flr_2 LENGTH->8 STARTBIT :48"}
Raw_X_T_Flr_2						:= _FB_CanRx_Message_Unpack_412.X_Byte_6;
GVL.IIVD.X_T_Flr_2.e				:= (Raw_X_T_Flr_2 > 16#FD) AND (Raw_X_T_Flr_2 < 16#FF);
GVL.IIVD.X_T_Flr_2.na				:= (Raw_X_T_Flr_2 = 16#FF);
GVL.IIVD.X_T_Flr_2.RangeExcd		:= NOT ((USINT_TO_REAL(BYTE_TO_USINT(Raw_X_T_Flr_2)) >= -40) AND (USINT_TO_REAL(BYTE_TO_USINT(Raw_X_T_Flr_2)) <= 100));
GVL.IIVD.X_T_Flr_2.v				:= NOT (_FB_CanRx_Message_Unpack_412.S_ER_TmOut OR GVL.IIVD.X_T_Flr_2.RangeExcd OR GVL.IIVD.X_T_Flr_2.e OR GVL.IIVD.X_T_Flr_2.na) ;
GVL.IIVD.X_T_Flr_2.x				:= 
(*SELECT 1 : Is data valid ?*)			SEL(GVL.IIVD.X_T_Flr_2.v,
(*DEFAULT value assigment*)				0,
(*Transmission is VALID*)				USINT_TO_REAL(BYTE_TO_USINT(Raw_X_T_Flr_2)) );
{endregion}

{region " SIGNAL AREA : NAME->W_T_Flr LENGTH->8 STARTBIT :56"}
Raw_W_T_Flr						:= _FB_CanRx_Message_Unpack_412.X_Byte_7;
GVL.IIVD.W_T_Flr.e					:= (Raw_W_T_Flr > 16#FD) AND (Raw_W_T_Flr < 16#FF);
GVL.IIVD.W_T_Flr.na					:= (Raw_W_T_Flr = 16#FF);
GVL.IIVD.W_T_Flr.RangeExcd			:= NOT ((USINT_TO_REAL(BYTE_TO_USINT(Raw_W_T_Flr)) >= -40) AND (USINT_TO_REAL(BYTE_TO_USINT(Raw_W_T_Flr)) <= 100));
GVL.IIVD.W_T_Flr.v					:= NOT (_FB_CanRx_Message_Unpack_412.S_ER_TmOut OR GVL.IIVD.W_T_Flr.RangeExcd OR GVL.IIVD.W_T_Flr.e OR GVL.IIVD.W_T_Flr.na) ;
GVL.IIVD.W_T_Flr.x					:= 
(*SELECT 1 : Is data valid ?*)			SEL(GVL.IIVD.W_T_Flr.v,
(*DEFAULT value assigment*)				0,
(*Transmission is VALID*)				USINT_TO_REAL(BYTE_TO_USINT(Raw_W_T_Flr)) );
{endregion}
{endregion}


GVL.IIVD.S_Com_Flt			:= 	GVL.IIVD.S_TmOut_Haberlesme_Durumlari_0X200 AND
								GVL.IIVD.S_TmOut_Direksiyon_Pompasi_Analog_0X210 AND
								GVL.IIVD.S_TmOut_Direksiyon_Pompasi_Durum_0X211 AND
								GVL.IIVD.S_TmOut_Arac_Durumlari_0X220 AND
								GVL.IIVD.S_TmOut_Fren_balata_durumlari_0X221 AND
								GVL.IIVD.S_TmOut_Fren_Basinclari_0X222 AND
								GVL.IIVD.S_TmOut_Lastik_Basinclari_1_0X223 AND
								GVL.IIVD.S_TmOut_Lastik_Basinclari_2_0X224 AND
								GVL.IIVD.S_TmOut_Arac_Bilgilendirme_0X225 AND
								GVL.IIVD.S_TmOut_Arac_Kritik_Uyarilari_0X226 AND
								GVL.IIVD.S_TmOut_Kapi_Hatalari_1_0X230 AND
								GVL.IIVD.S_TmOut_Kapi_Hatalari_2_0X231 AND
								GVL.IIVD.S_TmOut_Kapi_Hatalari_3_0X232 AND
								GVL.IIVD.S_TmOut_Kapi_Hatalari_4_0X233 AND
								GVL.IIVD.S_TmOut_Kapi_Hatalari_5_0X234 AND
								GVL.IIVD.S_TmOut_Kapi_Durum_1_0X235 AND
								GVL.IIVD.S_TmOut_Kapi_Durum_2_0X237 AND
								GVL.IIVD.S_TmOut_Kapi_Durum_3_0X238 AND
								GVL.IIVD.S_TmOut_Sigorta_Kontrol_1_0X260 AND
								GVL.IIVD.S_TmOut_Sigorta_Kontrol_2_0X261 AND
								GVL.IIVD.S_TmOut_Sigorta_Kontrol_3_0X262 AND
								GVL.IIVD.S_TmOut_Parametre_1_0X263 AND
// 								GVL.IIVD.S_TmOut_Diag_Temel_Durum_0X300 AND
// 								GVL.IIVD.S_TmOut_Diag_RTC_0X301 AND
// 								GVL.IIVD.S_TmOut_Diag_Parameter_0X302 AND
// 								GVL.IIVD.S_TmOut_Diag_Op_Rst_0X303 AND
// 								GVL.IIVD.S_TmOut_ECU_Dijital_Cikis_Test_0X310 AND
								GVL.IIVD.S_TmOut_Arac_Bilgi_2_0X2E1 AND
								GVL.IIVD.S_TmOut_Basamak_Isitici_Durumlari_0X412 AND TRUE;

GVL.IIVD.S_Com_Distrb		:= 	GVL.IIVD.S_TmOut_Haberlesme_Durumlari_0X200 OR
								GVL.IIVD.S_TmOut_Direksiyon_Pompasi_Analog_0X210 OR
								GVL.IIVD.S_TmOut_Direksiyon_Pompasi_Durum_0X211 OR
								GVL.IIVD.S_TmOut_Arac_Durumlari_0X220 OR
								GVL.IIVD.S_TmOut_Fren_balata_durumlari_0X221 OR
								GVL.IIVD.S_TmOut_Fren_Basinclari_0X222 OR
								GVL.IIVD.S_TmOut_Lastik_Basinclari_1_0X223 OR
								GVL.IIVD.S_TmOut_Lastik_Basinclari_2_0X224 OR
								GVL.IIVD.S_TmOut_Arac_Bilgilendirme_0X225 OR
								GVL.IIVD.S_TmOut_Arac_Kritik_Uyarilari_0X226 OR
								GVL.IIVD.S_TmOut_Kapi_Hatalari_1_0X230 OR
								GVL.IIVD.S_TmOut_Kapi_Hatalari_2_0X231 OR
								GVL.IIVD.S_TmOut_Kapi_Hatalari_3_0X232 OR
								GVL.IIVD.S_TmOut_Kapi_Hatalari_4_0X233 OR
								GVL.IIVD.S_TmOut_Kapi_Hatalari_5_0X234 OR
								GVL.IIVD.S_TmOut_Kapi_Durum_1_0X235 OR
								GVL.IIVD.S_TmOut_Kapi_Durum_2_0X237 OR
								GVL.IIVD.S_TmOut_Kapi_Durum_3_0X238 OR
								GVL.IIVD.S_TmOut_Sigorta_Kontrol_1_0X260 OR
								GVL.IIVD.S_TmOut_Sigorta_Kontrol_2_0X261 OR
								GVL.IIVD.S_TmOut_Sigorta_Kontrol_3_0X262 OR
								GVL.IIVD.S_TmOut_Parametre_1_0X263 OR
// 								GVL.IIVD.S_TmOut_Diag_Temel_Durum_0X300 OR
// 								GVL.IIVD.S_TmOut_Diag_RTC_0X301 OR
// 								GVL.IIVD.S_TmOut_Diag_Parameter_0X302 OR
// 								GVL.IIVD.S_TmOut_Diag_Op_Rst_0X303 OR
// 								GVL.IIVD.S_TmOut_ECU_Dijital_Cikis_Test_0X310 OR
								GVL.IIVD.S_TmOut_Arac_Bilgi_2_0X2E1 OR
								GVL.IIVD.S_TmOut_Basamak_Isitici_Durumlari_0X412 OR FALSE;


                  
END_PROGRAM

PROGRAM P_IOVD_A
  VAR
    N_Lf : USINT := 0;
    _FB_LfMon_0 : _FB_LfMon;
    _FB_CanTx_Message_Unpack_400 : _FB_CanTx_Message_Unpack;
    _FB_CanTx_Message_401 : _FB_CanTx_Message;
    _FB_CanTx_Message_402 : _FB_CanTx_Message;
    _FB_CanTx_Message_Unpack_450 : _FB_CanTx_Message_Unpack;
    _FB_CanTx_Message_Unpack_460 : _FB_CanTx_Message_Unpack;
    _FB_CanTx_Message_Unpack_462 : _FB_CanTx_Message_Unpack;
    _FB_CanTx_Message_463 : _FB_CanTx_Message;
    _FB_CanTx_Message_464 : _FB_CanTx_Message;
    _FB_CanTx_Message_465 : _FB_CanTx_Message;
    _FB_CanTx_Message_466 : _FB_CanTx_Message;
    _FB_CanTx_Message_467 : _FB_CanTx_Message;
    _FB_CanTx_Message_Unpack_480 : _FB_CanTx_Message_Unpack;
    _FB_CanTx_Message_Unpack_481 : _FB_CanTx_Message_Unpack;
    _FB_CanTx_Message_Unpack_482 : _FB_CanTx_Message_Unpack;
    _FB_CanTx_Message_Unpack_483 : _FB_CanTx_Message_Unpack;
    _FB_CanTx_Message_Unpack_484 : _FB_CanTx_Message_Unpack;
    _FB_CanTx_Message_Unpack_485 : _FB_CanTx_Message_Unpack;
    _FB_CanTx_Message_4C2 : _FB_CanTx_Message;
    _FB_CanTx_Message_Unpack_99 : _FB_CanTx_Message_Unpack;
    _FB_CanTx_Message_500 : _FB_CanTx_Message;
    _FB_UNPACK_DWORD_TO_BYTE_0 : _FB_UNPACK_DWORD_TO_BYTE;
    _FB_UNPACK_DWORD_TO_BYTE_1 : _FB_UNPACK_DWORD_TO_BYTE;
    _FB_UNPACK_WORD_TO_BYTE_0 : _FB_UNPACK_WORD_TO_BYTE;
    _FB_UNPACK_WORD_TO_BYTE_1 : _FB_UNPACK_WORD_TO_BYTE;
    _FB_UNPACK_WORD_TO_BYTE_2 : _FB_UNPACK_WORD_TO_BYTE;
    _FB_UNPACK_WORD_TO_BYTE_3 : _FB_UNPACK_WORD_TO_BYTE;
    _FB_UNPACK_WORD_TO_BYTE_4 : _FB_UNPACK_WORD_TO_BYTE;
    _FB_UNPACK_WORD_TO_BYTE_5 : _FB_UNPACK_WORD_TO_BYTE;
    _FB_UNPACK_WORD_TO_BYTE_6 : _FB_UNPACK_WORD_TO_BYTE;
    _FB_UNPACK_WORD_TO_BYTE_7 : _FB_UNPACK_WORD_TO_BYTE;
    _FB_UNPACK_WORD_TO_BYTE_8 : _FB_UNPACK_WORD_TO_BYTE;
    _FB_UNPACK_WORD_TO_BYTE_9 : _FB_UNPACK_WORD_TO_BYTE;
    _FB_UNPACK_WORD_TO_BYTE_10 : _FB_UNPACK_WORD_TO_BYTE;
    _FB_UNPACK_WORD_TO_BYTE_11 : _FB_UNPACK_WORD_TO_BYTE;
    _FB_UNPACK_WORD_TO_BYTE_12 : _FB_UNPACK_WORD_TO_BYTE;
    _FB_UNPACK_WORD_TO_BYTE_13 : _FB_UNPACK_WORD_TO_BYTE;
    _FB_UNPACK_WORD_TO_BYTE_14 : _FB_UNPACK_WORD_TO_BYTE;
    _FB_UNPACK_WORD_TO_BYTE_15 : _FB_UNPACK_WORD_TO_BYTE;
    _FB_UNPACK_WORD_TO_BYTE_16 : _FB_UNPACK_WORD_TO_BYTE;
    _FB_UNPACK_WORD_TO_BYTE_17 : _FB_UNPACK_WORD_TO_BYTE;
    _FB_UNPACK_WORD_TO_BYTE_18 : _FB_UNPACK_WORD_TO_BYTE;
    _FB_UNPACK_WORD_TO_BYTE_19 : _FB_UNPACK_WORD_TO_BYTE;
    _FB_UNPACK_WORD_TO_BYTE_20 : _FB_UNPACK_WORD_TO_BYTE;
    _FB_UNPACK_WORD_TO_BYTE_21 : _FB_UNPACK_WORD_TO_BYTE;
    _FB_UNPACK_WORD_TO_BYTE_22 : _FB_UNPACK_WORD_TO_BYTE;
    _FB_UNPACK_WORD_TO_BYTE_23 : _FB_UNPACK_WORD_TO_BYTE;
    _FB_UNPACK_WORD_TO_BYTE_24 : _FB_UNPACK_WORD_TO_BYTE;
    _FB_UNPACK_WORD_TO_BYTE_25 : _FB_UNPACK_WORD_TO_BYTE;
    _FB_UNPACK_WORD_TO_BYTE_26 : _FB_UNPACK_WORD_TO_BYTE;
    _FB_UNPACK_WORD_TO_BYTE_27 : _FB_UNPACK_WORD_TO_BYTE;
    _FB_UNPACK_WORD_TO_BYTE_28 : _FB_UNPACK_WORD_TO_BYTE;
    _FB_UNPACK_WORD_TO_BYTE_29 : _FB_UNPACK_WORD_TO_BYTE;
    _FB_UNPACK_WORD_TO_BYTE_30 : _FB_UNPACK_WORD_TO_BYTE;
    _FB_UNPACK_BYTE_TO_8BITS_0 : _FB_UNPACK_BYTE_TO_8BITS;
    _FB_UNPACK_BYTE_TO_8BITS_1 : _FB_UNPACK_BYTE_TO_8BITS;
    _FB_UNPACK_BYTE_TO_8BITS_2 : _FB_UNPACK_BYTE_TO_8BITS;
    _FB_PACK_8BITS_TO_BYTE_0 : _FB_PACK_8BITS_TO_BYTE;
    _FB_PACK_8BITS_TO_BYTE_1 : _FB_PACK_8BITS_TO_BYTE;
    _FB_PACK_8BITS_TO_BYTE_2 : _FB_PACK_8BITS_TO_BYTE;
    _FB_PACK_8BITS_TO_BYTE_3 : _FB_PACK_8BITS_TO_BYTE;
    _FB_PACK_8BITS_TO_BYTE_4 : _FB_PACK_8BITS_TO_BYTE;
    _FB_PACK_8BITS_TO_BYTE_5 : _FB_PACK_8BITS_TO_BYTE;
    _FB_PACK_8BITS_TO_BYTE_6 : _FB_PACK_8BITS_TO_BYTE;
    _FB_PACK_8BITS_TO_BYTE_7 : _FB_PACK_8BITS_TO_BYTE;
    T_TCU_Mjr : BOOL := FALSE;
    T_TCU_Mnr : BOOL := FALSE;
    T_TCU_Flt : BOOL := FALSE;
  END_VAR

                    (*
**********************************************************************
Bozankaya A.Ş.
**********************************************************************
Name					: P_IOVD_A
POU Type				: Program
Created by              : COMMUNICATION INTERFACE GENERATOR V1.1.034(denizcikispc), BZK.
Creation Date 			: 2023-07-11T10:31:49
Modifications			: see version description below


Program Description:This program which is created by automatically by communication interface generator 
 handles the TX (OUTPUT) can messages according to CAN_500_LIB 
*********************************************************************

Version 1	
*********************************************************************
Version Description:
- initial version
*********************************************************************
*)
//-----------------------------------------------------------------------------------------------------------------------------
//MESSAGE------
{region " User Area : ECU_Haberlesme- ID:400"}

Bazı kısımları sildim ve bu yazıyı ekliyorum
//-------SIGNAL -> S_ER_Com_ESS Max: 1 Min: 0 Def: 0 Resolution: 1 Offset: 0
GVL.IOVD.S_ER_Com_ESS.v						:= GVL.SY.S_ECU_Rdy AND NOT GVL.IOVD.S_ER_Com_ESS.e AND NOT GVL.IOVD.S_ER_Com_ESS.na;
GVL.IOVD.S_ER_Com_ESS.x						:= GVL.IIME.S_Com_Distrb;
GVL.IOVD.S_ER_Com_ESS.e						:= FALSE;
GVL.IOVD.S_ER_Com_ESS.na					:= FALSE;
//-------SIGNAL -> S_ER_Com_HVAC Max: 1 Min: 0 Def: 0 Resolution: 1 Offset: 0
GVL.IOVD.S_ER_Com_HVAC.v					:= GVL.SY.S_ECU_Rdy AND NOT GVL.IOVD.S_ER_Com_HVAC.e AND NOT GVL.IOVD.S_ER_Com_HVAC.na;
GVL.IOVD.S_ER_Com_HVAC.x					:= GVL.IICH.S_Com_Distrb;
GVL.IOVD.S_ER_Com_HVAC.e					:= FALSE;
GVL.IOVD.S_ER_Com_HVAC.na					:= FALSE;
//-------SIGNAL -> S_ER_Com_EBS Max: 1 Min: 0 Def: 0 Resolution: 1 Offset: 0
GVL.IOVD.S_ER_Com_EBS.v						:= GVL.SY.S_ECU_Rdy AND NOT GVL.IOVD.S_ER_Com_EBS.e AND NOT GVL.IOVD.S_ER_Com_EBS.na;
GVL.IOVD.S_ER_Com_EBS.x						:= GVL.IIBA.S_Com_Distrb;
GVL.IOVD.S_ER_Com_EBS.e						:= FALSE;
GVL.IOVD.S_ER_Com_EBS.na					:= FALSE;
//-------SIGNAL -> S_ER_Com_PCAN Max: 1 Min: 0 Def: 0 Resolution: 1 Offset: 0
GVL.IOVD.S_ER_Com_PCAN.v					:= GVL.SY.S_ECU_Rdy AND NOT GVL.IOVD.S_ER_Com_PCAN.e AND NOT GVL.IOVD.S_ER_Com_PCAN.na;
GVL.IOVD.S_ER_Com_PCAN.x					:= GVL.VD.S_PCAN_Flt;
GVL.IOVD.S_ER_Com_PCAN.e					:= FALSE;
GVL.IOVD.S_ER_Com_PCAN.na					:= FALSE;
//-------SIGNAL -> S_ER_Com_Pnt Max: 1 Min: 0 Def: 0 Resolution: 1 Offset: 0
GVL.IOVD.S_ER_Com_Pnt.v						:= GVL.SY.S_ECU_Rdy AND NOT GVL.IOVD.S_ER_Com_Pnt.e AND NOT GVL.IOVD.S_ER_Com_Pnt.na;
GVL.IOVD.S_ER_Com_Pnt.x						:= GVL.IIMP.S_Com_Distrb;
GVL.IOVD.S_ER_Com_Pnt.e						:= FALSE;
GVL.IOVD.S_ER_Com_Pnt.na					:= FALSE;
//-------SIGNAL -> S_ER_Com_Acc_Pdl Max: 1 Min: 0 Def: 0 Resolution: 1 Offset: 0
GVL.IOVD.S_ER_Com_Acc_Pdl.v					:= GVL.SY.S_ECU_Rdy AND NOT GVL.IOVD.S_ER_Com_Acc_Pdl.e AND NOT GVL.IOVD.S_ER_Com_Acc_Pdl.na;
GVL.IOVD.S_ER_Com_Acc_Pdl.x					:= GVL.IIPA.S_Com_Distrb;
GVL.IOVD.S_ER_Com_Acc_Pdl.e					:= FALSE;
GVL.IOVD.S_ER_Com_Acc_Pdl.na				:= FALSE;
//-------SIGNAL -> S_ER_Com_Str_Ang_Snsr Max: 1 Min: 0 Def: 0 Resolution: 1 Offset: 0
GVL.IOVD.S_ER_Com_Str_Ang_Snsr.v			:= GVL.SY.S_ECU_Rdy AND NOT GVL.IOVD.S_ER_Com_Str_Ang_Snsr.e AND NOT GVL.IOVD.S_ER_Com_Str_Ang_Snsr.na;
GVL.IOVD.S_ER_Com_Str_Ang_Snsr.x			:= GVL.IIRS.S_Com_Distrb;
GVL.IOVD.S_ER_Com_Str_Ang_Snsr.e			:= FALSE;
GVL.IOVD.S_ER_Com_Str_Ang_Snsr.na 			:= FALSE;
//-------SIGNAL -> S_PDU_Cvr_Op Max: 1 Min: 0 Def: 0 Resolution: 1 Offset: 0
GVL.IOVD.S_PDU_Cvr_Op.v						:= GVL.SY.S_ECU_Rdy AND NOT GVL.IOVD.S_PDU_Cvr_Op.e AND NOT GVL.IOVD.S_PDU_Cvr_Op.na;
GVL.IOVD.S_PDU_Cvr_Op.x						:=  NOT GVL.IIRE.S_PDU_Cvr_Cl.pin_value;
GVL.IOVD.S_PDU_Cvr_Op.e						:= FALSE;
GVL.IOVD.S_PDU_Cvr_Op.na					:= FALSE;			   

//-------SIGNAL -> S_ER_HVAC_Red Max: 1 Min: 0 Def: 0 Resolution: 1 Offset: 0
GVL.IOVD.S_ER_HVAC_Red.v					:= GVL.SY.S_ECU_Rdy;
GVL.IOVD.S_ER_HVAC_Red.x					:= FALSE;
//-------SIGNAL -> S_ER_Iso_Amb Max: 1 Min: 0 Def: 0 Resolution: 1 Offset: 0
GVL.IOVD.S_ER_Iso_Amb.v						:= GVL.SY.S_ECU_Rdy;
GVL.IOVD.S_ER_Iso_Amb.x						:= GVL.PI.S_Err_Insu_Flt_Amb;
//-------SIGNAL -> S_ER_Iso_Red Max: 1 Min: 0 Def: 0 Resolution: 1 Offset: 0
GVL.IOVD.S_ER_Iso_Red.v						:= GVL.SY.S_ECU_Rdy;
GVL.IOVD.S_ER_Iso_Red.x						:= GVL.PI.S_Err_Insu_Flt_Red;
//-------SIGNAL -> S_ER_Amb Max: 1 Min: 0 Def: 0 Resolution: 1 Offset: 0
GVL.IOVD.S_ER_Amb.v							:= GVL.SY.S_ECU_Rdy;
GVL.IOVD.S_ER_Amb.x							:= GVL.VD.S_Err_Amb;
//-------SIGNAL -> S_ER_Red Max: 1 Min: 0 Def: 0 Resolution: 1 Offset: 0
GVL.IOVD.S_ER_Red.v							:= GVL.SY.S_ECU_Rdy;
GVL.IOVD.S_ER_Red.x							:= GVL.VD.S_Err_Red;
//-------SIGNAL -> S_Rdy_Dep Max: 1 Min: 0 Def: 0 Resolution: 1 Offset: 0
GVL.IOVD.S_Rdy_Dep.v						:= GVL.SY.S_ECU_Rdy;
//-------SIGNAL -> S_Pwr_Red Max: 1 Min: 0 Def: 0 Resolution: 1 Offset: 0
GVL.IOVD.S_Pwr_Red.v						:= GVL.SY.S_ECU_Rdy;
GVL.IOVD.S_Pwr_Red.x						:= GVL.ME.S_Err_Bat_Pckt_Onl OR GVL.ME.S_Err_Dischrg_Curr_Rdc;
//-------SIGNAL -> S_ER_BCU_Amb Max: 1 Min: 0 Def: 0 Resolution: 1 Offset: 0
GVL.IOVD.S_ER_BCU_Amb.v						:= GVL.SY.S_ECU_Rdy;
GVL.IOVD.S_ER_BCU_Amb.x						:= NOT GVL.IIBA.S_ABS_Full_Op.x OR GVL.IIBA.S_EBS_ABS_Amb_Wrn.x;
//-------SIGNAL -> S_ER_BCU_Red Max: 1 Min: 0 Def: 0 Resolution: 1 Offset: 0
GVL.IOVD.S_ER_BCU_Red.v						:= GVL.SY.S_ECU_Rdy;
GVL.IOVD.S_ER_BCU_Red.x						:= GVL.IIBA.S_EBS_Red_Wrn.x;
//-------SIGNAL -> S_ER_Temp_Red Max: 1 Min: 0 Def: 0 Resolution: 1 Offset: 0
GVL.IOVD.S_ER_Temp_Red.v					:= GVL.SY.S_ECU_Rdy;
// GVL.IOVD.S_ER_Temp_Red.x					:= FALSE;
//-------SIGNAL -> S_ER_Temp_Amb Max: 1 Min: 0 Def: 0 Resolution: 1 Offset: 0
GVL.IOVD.S_ER_Temp_Amb.v					:= GVL.SY.S_ECU_Rdy;
// GVL.IOVD.S_ER_Temp_Amb.x					:= FALSE;
//-------SIGNAL -> S_ER_HV_Amb Max: 1 Min: 0 Def: 0 Resolution: 1 Offset: 0
GVL.IOVD.S_ER_HV_Amb.v						:= GVL.SY.S_ECU_Rdy;
GVL.IOVD.S_ER_HV_Amb.x						:= GVL.ME.S_Err_HV_Amb;
// PR1006_SRS_001181_TIMTRO 
//-------SIGNAL -> S_ER_HV_Red Max: 1 Min: 0 Def: 0 Resolution: 1 Offset: 0
GVL.IOVD.S_ER_HV_Red.v						:= GVL.SY.S_ECU_Rdy;
GVL.IOVD.S_ER_HV_Red.x						:= GVL.ME.S_Err_HV_Red;
//-------SIGNAL -> S_ER_Pnt_Amb Max: 1 Min: 0 Def: 0 Resolution: 1 Offset: 0
GVL.IOVD.S_ER_Pnt_Amb.v						:= GVL.SY.S_ECU_Rdy;
GVL.IOVD.S_ER_Pnt_Amb.x						:= GVL.MP.S_Err_Pnt_Amb;
//-------SIGNAL -> S_ER_Pnt_Red Max: 1 Min: 0 Def: 0 Resolution: 1 Offset: 0
GVL.IOVD.S_ER_Pnt_Red.v						:= GVL.SY.S_ECU_Rdy;
GVL.IOVD.S_ER_Pnt_Red.x						:= GVL.MP.S_Err_Pnt_Red;
//-------SIGNAL -> S_Mot_Temp_Hi Max: 1 Min: 0 Def: 0 Resolution: 1 Offset: 0
GVL.IOVD.S_Mot_Temp_Hi.v					:= GVL.SY.S_ECU_Rdy;
// GVL.IOVD.S_Mot_Temp_Hi.x					:= FALSE;
//-------SIGNAL -> S_Mot_Temp_Too_Hi Max: 1 Min: 0 Def: 0 Resolution: 1 Offset: 0
GVL.IOVD.S_Mot_Temp_Too_Hi.v				:= GVL.SY.S_ECU_Rdy;
// GVL.IOVD.S_Mot_Temp_Too_Hi.x				:= FALSE;
//-------SIGNAL -> S_ER_BCCU Max: 1 Min: 0 Def: 0 Resolution: 1 Offset: 0
GVL.IOVD.S_ER_BCCU.v						:= GVL.SY.S_ECU_Rdy;
GVL.IOVD.S_ER_BCCU.x						:= FALSE;
//-------SIGNAL -> S_Ln_Vo_Lo Max: 1 Min: 0 Def: 0 Resolution: 1 Offset: 0
GVL.IOVD.S_Ln_Vo_Lo.v						:= GVL.SY.S_ECU_Rdy;
GVL.IOVD.S_Ln_Vo_Lo.x						:= GVL.MP.S_Err_Cat_Ln_Volt_Lo;
//-------SIGNAL -> S_Ln_Vo_Too_Lo Max: 1 Min: 0 Def: 0 Resolution: 1 Offset: 0
GVL.IOVD.S_Ln_Vo_Hi.v						:= GVL.SY.S_ECU_Rdy;
GVL.IOVD.S_Ln_Vo_Hi.x						:= GVL.MP.S_Err_Cat_Ln_Volt_Hi;
//-------SIGNAL -> S_ER_Mot_Cnv_Amb Max: 1 Min: 0 Def: 0 Resolution: 1 Offset: 0
GVL.IOVD.S_ER_Mot_Cnv_Amb.v					:= GVL.SY.S_ECU_Rdy;
GVL.IOVD.S_ER_Mot_Cnv_Amb.x					:= FALSE;
//-------SIGNAL -> S_ER_Mot_Cnv_Red Max: 1 Min: 0 Def: 0 Resolution: 1 Offset: 0
GVL.IOVD.S_ER_Mot_Cnv_Red.v					:= GVL.SY.S_ECU_Rdy;
GVL.IOVD.S_ER_Mot_Cnv_Red.x					:= FALSE;
//-------SIGNAL -> S_ER_Icy_Road_Amb Max: 1 Min: 0 Def: 0 Resolution: 1 Offset: 0
GVL.IOVD.S_ER_Icy_Road_Amb.v				:= GVL.SY.S_ECU_Rdy;
// GVL.IOVD.S_ER_Icy_Road_Amb.x				:= FALSE;
//-------SIGNAL -> S_ER_Str_Pmp_Temp_Hi Max: 1 Min: 0 Def: 0 Resolution: 1 Offset: 0
GVL.IOVD.S_ER_Str_Pmp_Temp_Hi.v				:= GVL.SY.S_ECU_Rdy;
// GVL.IOVD.S_ER_Str_Pmp_Temp_Hi.x			:= FALSE;
//-------SIGNAL -> S_ER_Aux_AC_Amb Max: 1 Min: 0 Def: 0 Resolution: 1 Offset: 0
GVL.IOVD.S_ER_Aux_AC_Amb.v					:= GVL.SY.S_ECU_Rdy;
GVL.IOVD.S_ER_Aux_AC_Amb.x					:= FALSE;
//-------SIGNAL -> S_ER_Aux_AC_Red Max: 1 Min: 0 Def: 0 Resolution: 1 Offset: 0
GVL.IOVD.S_ER_Aux_AC_Red.v					:= GVL.SY.S_ECU_Rdy;
GVL.IOVD.S_ER_Aux_AC_Red.x					:= FALSE;
//-------SIGNAL -> Vehicle_mode_bitmask Max: 255 Min: 0 Def: 0 Resolution: 1 Offset: 0
GVL.IOVD.Z_Vh_Mode.v					:= GVL.SY.S_ECU_Rdy AND NOT GVL.IOVD.Z_Vh_Mode.e AND NOT GVL.IOVD.Z_Vh_Mode.na AND NOT GVL.IOVD.Z_Vh_Mode.RangeExcd;

_FB_PACK_8BITS_TO_BYTE_1 (	S_BIT_0 	:= GVL.IIPT.S_Bat_Mod_Stat.x,
						 	S_BIT_1		:= GVL.IIPT.S_Trol_Mod_Actv.x,
						 	S_BIT_2 	:= GVL.MC.S_Inlt_Conn,
						 	S_BIT_3 	:= 0,
						 	S_BIT_4 	:= GVL.IIPT.X_I_DCDC_Out.x <> 0,
						 	S_BIT_5 	:= 0, //Force/Test mode
						 	S_BIT_6 	:= GVL.MR.S_Em_Stop,
						 	S_BIT_7 	:= 0,
						 	X_BYTE_0 	=> GVL.IOVD.Z_Vh_Mode.x);

GVL.IOVD.Z_Vh_Mode.e						:= FALSE;
GVL.IOVD.Z_Vh_Mode.na						:= FALSE;
GVL.IOVD.Z_Vh_Mode.RangeExcd				:=  (255 < GVL.IOVD.Z_Vh_Mode.x) OR (0 > GVL.IOVD.Z_Vh_Mode.x);
{endregion}
//-----------------------------------------------------------------------------------------------------------------------------
//-----------------------------------------------------------------------------------------------------------------------------
//MESSAGE------
{region " User Area : DDS- ID:401"}
//-------SIGNAL -> X_DDS_No_1 Max: 65535 Min: 0 Def: 0 Resolution: 1 Offset: 0
GVL.IOVD.X_DDS_No_1.v					:= GVL.SY.S_ECU_Rdy AND NOT GVL.IOVD.X_DDS_No_1.e AND NOT GVL.IOVD.X_DDS_No_1.na AND NOT GVL.IOVD.X_DDS_No_1.RangeExcd;
GVL.IOVD.X_DDS_No_1.e					:= FALSE;
GVL.IOVD.X_DDS_No_1.na					:= FALSE;
GVL.IOVD.X_DDS_No_1.RangeExcd			:=  (65535 < GVL.IOVD.X_DDS_No_1.x )OR (0 > GVL.IOVD.X_DDS_No_1.x);
//-------SIGNAL -> X_DDS_No_2 Max: 65535 Min: 0 Def: 0 Resolution: 1 Offset: 0
GVL.IOVD.X_DDS_No_2.v					:= GVL.SY.S_ECU_Rdy AND NOT GVL.IOVD.X_DDS_No_2.e AND NOT GVL.IOVD.X_DDS_No_2.na AND NOT GVL.IOVD.X_DDS_No_2.RangeExcd;
GVL.IOVD.X_DDS_No_2.e					:= FALSE;
GVL.IOVD.X_DDS_No_2.na					:= FALSE;
GVL.IOVD.X_DDS_No_2.RangeExcd			:=  (65535 < GVL.IOVD.X_DDS_No_2.x )OR (0 > GVL.IOVD.X_DDS_No_2.x);
//-------SIGNAL -> X_DDS_No_3 Max: 65535 Min: 0 Def: 0 Resolution: 1 Offset: 0
GVL.IOVD.X_DDS_No_3.v					:= GVL.SY.S_ECU_Rdy AND NOT GVL.IOVD.X_DDS_No_3.e AND NOT GVL.IOVD.X_DDS_No_3.na AND NOT GVL.IOVD.X_DDS_No_3.RangeExcd;
GVL.IOVD.X_DDS_No_3.e					:= FALSE;
GVL.IOVD.X_DDS_No_3.na					:= FALSE;
GVL.IOVD.X_DDS_No_3.RangeExcd			:=  (65535 < GVL.IOVD.X_DDS_No_3.x )OR (0 > GVL.IOVD.X_DDS_No_3.x);
//-------SIGNAL -> X_DDS_No_4 Max: 65535 Min: 0 Def: 0 Resolution: 1 Offset: 0
GVL.IOVD.X_DDS_No_4.v					:= GVL.SY.S_ECU_Rdy AND NOT GVL.IOVD.X_DDS_No_4.e AND NOT GVL.IOVD.X_DDS_No_4.na AND NOT GVL.IOVD.X_DDS_No_4.RangeExcd;
GVL.IOVD.X_DDS_No_4.e					:= FALSE;
GVL.IOVD.X_DDS_No_4.na					:= FALSE;
GVL.IOVD.X_DDS_No_4.RangeExcd			:=  (65535 < GVL.IOVD.X_DDS_No_4.x )OR (0 > GVL.IOVD.X_DDS_No_4.x);
{endregion}
//-----------------------------------------------------------------------------------------------------------------------------
//-----------------------------------------------------------------------------------------------------------------------------
//MESSAGE------
{region " User Area : DDS_2- ID:402"}
//-------SIGNAL -> X_DDS_No_5 Max: 65535 Min: 0 Def: 0 Resolution: 1 Offset: 0
GVL.IOVD.X_DDS_No_5.v					:= GVL.SY.S_ECU_Rdy AND NOT GVL.IOVD.X_DDS_No_5.e AND NOT GVL.IOVD.X_DDS_No_5.na AND NOT GVL.IOVD.X_DDS_No_5.RangeExcd;
GVL.IOVD.X_DDS_No_5.e					:= FALSE;
GVL.IOVD.X_DDS_No_5.na					:= FALSE;
GVL.IOVD.X_DDS_No_5.RangeExcd			:=  (65535 < GVL.IOVD.X_DDS_No_5.x )OR (0 > GVL.IOVD.X_DDS_No_5.x);
//-------SIGNAL -> X_Tot_Pg_No Max: 255 Min: 0 Def: 0 Resolution: 1 Offset: 0
GVL.IOVD.X_Tot_Pg_No.v					:= GVL.SY.S_ECU_Rdy AND NOT GVL.IOVD.X_Tot_Pg_No.e AND NOT GVL.IOVD.X_Tot_Pg_No.na AND NOT GVL.IOVD.X_Tot_Pg_No.RangeExcd;
GVL.IOVD.X_Tot_Pg_No.e					:= FALSE;
GVL.IOVD.X_Tot_Pg_No.na					:= FALSE;
GVL.IOVD.X_Tot_Pg_No.RangeExcd			:=  (255 < GVL.IOVD.X_Tot_Pg_No.x )OR (0 > GVL.IOVD.X_Tot_Pg_No.x);
//-------SIGNAL -> X_Cur_Pg_No Max: 255 Min: 0 Def: 0 Resolution: 1 Offset: 0
GVL.IOVD.X_Cur_Pg_No.v					:= GVL.SY.S_ECU_Rdy AND NOT GVL.IOVD.X_Cur_Pg_No.e AND NOT GVL.IOVD.X_Cur_Pg_No.na AND NOT GVL.IOVD.X_Cur_Pg_No.RangeExcd;
GVL.IOVD.X_Cur_Pg_No.e					:= FALSE;
GVL.IOVD.X_Cur_Pg_No.na					:= FALSE;
GVL.IOVD.X_Cur_Pg_No.RangeExcd			:=  (255 < GVL.IOVD.X_Cur_Pg_No.x )OR (0 > GVL.IOVD.X_Cur_Pg_No.x);
{endregion}
//-----------------------------------------------------------------------------------------------------------------------------
//-----------------------------------------------------------------------------------------------------------------------------
//MESSAGE------
{region " User Area : HV_Durum- ID:450"}

//-------SIGNAL -> C_Ign_Hv_On Max: 1 Min: 0 Def: 0 Resolution: 1 Offset: 0

//-------SIGNAL -> C_Ign_Hv_On Max: 1 Min: 0 Def: 0 Resolution: 1 Offset: 0
GVL.IOVD.C_Ign_Hv_On.v						:= GVL.SY.S_ECU_Rdy AND NOT GVL.IOVD.C_Ign_Hv_On.e AND NOT GVL.IOVD.C_Ign_Hv_On.na;
GVL.IOVD.C_Ign_Hv_On.x						:= GVL.ME.C_Ign_HV_On;
GVL.IOVD.C_Ign_Hv_On.e						:= FALSE;
GVL.IOVD.C_Ign_Hv_On.na						:= FALSE;
//-------SIGNAL -> C_Pnt_Hv_On Max: 1 Min: 0 Def: 0 Resolution: 1 Offset: 0
GVL.IOVD.C_Pnt_Hv_On.v						:= GVL.SY.S_ECU_Rdy AND NOT GVL.IOVD.C_Pnt_Hv_On.e AND NOT GVL.IOVD.C_Pnt_Hv_On.na;
GVL.IOVD.C_Pnt_Hv_On.x						:= FALSE;
GVL.IOVD.C_Pnt_Hv_On.e						:= FALSE;
GVL.IOVD.C_Pnt_Hv_On.na						:= FALSE;
//-------SIGNAL -> C_Bat_Lo_Hv_On Max: 1 Min: 0 Def: 0 Resolution: 1 Offset: 0
GVL.IOVD.C_Bat_Lo_Hv_On.v					:= GVL.SY.S_ECU_Rdy AND NOT GVL.IOVD.C_Bat_Lo_Hv_On.e AND NOT GVL.IOVD.C_Bat_Lo_Hv_On.na;
GVL.IOVD.C_Bat_Lo_Hv_On.x					:= GVL.ME.C_Lo_24V_HV_On OR NOT GVL.SY.S_B2_On;
GVL.IOVD.C_Bat_Lo_Hv_On.e					:= FALSE;
GVL.IOVD.C_Bat_Lo_Hv_On.na					:= FALSE;
//-------SIGNAL -> C_Tm_Hv_On Max: 1 Min: 0 Def: 0 Resolution: 1 Offset: 0
GVL.IOVD.C_Tm_Hv_On.v						:= GVL.SY.S_ECU_Rdy AND NOT GVL.IOVD.C_Tm_Hv_On.e AND NOT GVL.IOVD.C_Tm_Hv_On.na;
GVL.IOVD.C_Tm_Hv_On.x						:= GVL.ME.C_Tm_HV_On;
GVL.IOVD.C_Tm_Hv_On.e						:= FALSE;
GVL.IOVD.C_Tm_Hv_On.na						:= FALSE;
//-------SIGNAL -> C_Diag_Hv_On Max: 1 Min: 0 Def: 0 Resolution: 1 Offset: 0
GVL.IOVD.C_Diag_Hv_On.v						:= GVL.SY.S_ECU_Rdy AND NOT GVL.IOVD.C_Diag_Hv_On.e AND NOT GVL.IOVD.C_Diag_Hv_On.na;
GVL.IOVD.C_Diag_Hv_On.x						:= GVL.ME.C_Diag_HV_On;
GVL.IOVD.C_Diag_Hv_On.e						:= FALSE;
GVL.IOVD.C_Diag_Hv_On.na					:= FALSE;
//-------SIGNAL -> C_Ign_Hv_Off Max: 1 Min: 0 Def: 0 Resolution: 1 Offset: 0
GVL.IOVD.C_Ign_Hv_Off.v						:= GVL.SY.S_ECU_Rdy AND NOT GVL.IOVD.C_Ign_Hv_Off.e AND NOT GVL.IOVD.C_Ign_Hv_Off.na;
GVL.IOVD.C_Ign_Hv_Off.x						:= NOT GVL.ME.C_Ign_HV_On;
GVL.IOVD.C_Ign_Hv_Off.e						:= FALSE;
GVL.IOVD.C_Ign_Hv_Off.na					:= FALSE;
//-------SIGNAL -> C_Pnt_Hv_Off Max: 1 Min: 0 Def: 0 Resolution: 1 Offset: 0
GVL.IOVD.C_Pnt_Hv_Off.v						:= GVL.SY.S_ECU_Rdy AND NOT GVL.IOVD.C_Pnt_Hv_Off.e AND NOT GVL.IOVD.C_Pnt_Hv_Off.na;
GVL.IOVD.C_Pnt_Hv_Off.x						:= FALSE;
GVL.IOVD.C_Pnt_Hv_Off.e						:= FALSE;
GVL.IOVD.C_Pnt_Hv_Off.na					:= FALSE;
//-------SIGNAL -> C_Bat_Lo_Hv_Off Max: 1 Min: 0 Def: 0 Resolution: 1 Offset: 0
GVL.IOVD.C_Bat_Lo_Hv_Off.v					:= GVL.SY.S_ECU_Rdy AND NOT GVL.IOVD.C_Bat_Lo_Hv_Off.e AND NOT GVL.IOVD.C_Bat_Lo_Hv_Off.na;
GVL.IOVD.C_Bat_Lo_Hv_Off.x					:= NOT GVL.ME.C_Lo_24V_HV_On;
GVL.IOVD.C_Bat_Lo_Hv_Off.e					:= FALSE;
GVL.IOVD.C_Bat_Lo_Hv_Off.na					:= FALSE;
//-------SIGNAL -> C_Tm_Hv_Off Max: 1 Min: 0 Def: 0 Resolution: 1 Offset: 0
GVL.IOVD.C_Tm_Hv_Off.v						:= GVL.SY.S_ECU_Rdy AND NOT GVL.IOVD.C_Tm_Hv_Off.e AND NOT GVL.IOVD.C_Tm_Hv_Off.na;
GVL.IOVD.C_Tm_Hv_Off.x						:= NOT GVL.ME.C_Tm_HV_On;
GVL.IOVD.C_Tm_Hv_Off.e						:= FALSE;
GVL.IOVD.C_Tm_Hv_Off.na						:= FALSE;
//-------SIGNAL -> C_Diag_Hv_Off Max: 1 Min: 0 Def: 0 Resolution: 1 Offset: 0
GVL.IOVD.C_Diag_Hv_Off.v					:= GVL.SY.S_ECU_Rdy AND NOT GVL.IOVD.C_Diag_Hv_Off.e AND NOT GVL.IOVD.C_Diag_Hv_Off.na;
GVL.IOVD.C_Diag_Hv_Off.x					:= NOT GVL.ME.C_Diag_HV_On;
GVL.IOVD.C_Diag_Hv_Off.e					:= FALSE;
GVL.IOVD.C_Diag_Hv_Off.na					:= FALSE;
//-------SIGNAL -> C_Hv_On Max: 1 Min: 0 Def: 0 Resolution: 1 Offset: 0
GVL.IOVD.C_Hv_On.v							:= GVL.SY.S_ECU_Rdy AND NOT GVL.IOVD.C_Hv_On.e AND NOT GVL.IOVD.C_Hv_On.na;
GVL.IOVD.C_Hv_On.x							:= GVL.ME.C_HV_On;
GVL.IOVD.C_Hv_On.e							:= FALSE;
GVL.IOVD.C_Hv_On.na							:= FALSE;
//-------SIGNAL -> C_Hv_Off Max: 1 Min: 0 Def: 0 Resolution: 1 Offset: 0
GVL.IOVD.C_Hv_Off.v							:= GVL.SY.S_ECU_Rdy AND NOT GVL.IOVD.C_Hv_Off.e AND NOT GVL.IOVD.C_Hv_Off.na;
GVL.IOVD.C_Hv_Off.x							:= NOT GVL.ME.C_HV_On;
GVL.IOVD.C_Hv_Off.e							:= FALSE;
GVL.IOVD.C_Hv_Off.na						:= FALSE;
//-------SIGNAL -> S_Hv_On_Prc Max: 1 Min: 0 Def: 0 Resolution: 1 Offset: 0
GVL.IOVD.S_Hv_On_Prc.v						:= GVL.SY.S_ECU_Rdy AND NOT GVL.IOVD.S_Hv_On_Prc.e AND NOT GVL.IOVD.S_Hv_On_Prc.na;
GVL.IOVD.S_Hv_On_Prc.x						:= GVL.ME.X_Stat_No > 10 AND GVL.ME.X_Stat_No < 50;
GVL.IOVD.S_Hv_On_Prc.e						:= FALSE;
GVL.IOVD.S_Hv_On_Prc.na						:= FALSE;
//-------SIGNAL -> S_Hv_Off_Prc Max: 1 Min: 0 Def: 0 Resolution: 1 Offset: 0
GVL.IOVD.S_Hv_Off_Prc.v						:= GVL.SY.S_ECU_Rdy AND NOT GVL.IOVD.S_Hv_Off_Prc.e AND NOT GVL.IOVD.S_Hv_Off_Prc.na;
GVL.IOVD.S_Hv_Off_Prc.x						:= GVL.ME.X_Stat_No > 50 AND GVL.ME.X_Stat_No < 75;
GVL.IOVD.S_Hv_Off_Prc.e						:= FALSE;
GVL.IOVD.S_Hv_Off_Prc.na					:= FALSE;
//-------SIGNAL -> S_Em_Stop Max: 1 Min: 0 Def: 0 Resolution: 1 Offset: 0
GVL.IOVD.S_Em_Stop.v						:= GVL.SY.S_ECU_Rdy AND NOT GVL.IOVD.S_Em_Stop.e AND NOT GVL.IOVD.S_Em_Stop.na;
GVL.IOVD.S_Em_Stop.x						:= GVL.MR.S_Em_Stop;
GVL.IOVD.S_Em_Stop.e						:= FALSE;
GVL.IOVD.S_Em_Stop.na						:= FALSE;
//-------SIGNAL -> S_Hv_On_En Max: 1 Min: 0 Def: 0 Resolution: 1 Offset: 0
GVL.IOVD.S_Hv_On_En.v						:= GVL.SY.S_ECU_Rdy AND NOT GVL.IOVD.S_Hv_Off_Prc.e AND NOT GVL.IOVD.S_Hv_Off_Prc.na;
GVL.IOVD.S_Hv_On_En.x						:= GVL.ME.S_HV_On_Sfty_Cond_Ok AND (GVL.ME.C_Ign_HV_On OR GVL.ME.S_Trol_Mod_HV_Req);
GVL.IOVD.S_Hv_On_En.e						:= FALSE;
GVL.IOVD.S_Hv_On_En.na						:= FALSE;
//-------SIGNAL -> S_Hv_Off_En Max: 1 Min: 0 Def: 0 Resolution: 1 Offset: 0
GVL.IOVD.S_Hv_Off_En.v						:= GVL.SY.S_ECU_Rdy AND NOT GVL.IOVD.S_Hv_Off_Prc.e AND NOT GVL.IOVD.S_Hv_Off_Prc.na;
GVL.IOVD.S_Hv_Off_En.x						:= GVL.ME.S_HV_Off_Sfty_Cond_Ok;
GVL.IOVD.S_Hv_Off_En.e						:= FALSE;
GVL.IOVD.S_Hv_Off_En.na						:= FALSE;
//-------SIGNAL -> C_Mn_Ct_On Max: 1 Min: 0 Def: 0 Resolution: 1 Offset: 0
GVL.IOVD.C_Mn_Ct_On.v						:= GVL.SY.S_ECU_Rdy AND NOT GVL.IOVD.C_Mn_Ct_On.e AND NOT GVL.IOVD.C_Mn_Ct_On.na;
GVL.IOVD.C_Mn_Ct_On.x						:= GVL.IOME.C_Mn_Ct.x;
GVL.IOVD.C_Mn_Ct_On.e						:= GVL.IOME.C_Mn_Ct.e;
GVL.IOVD.C_Mn_Ct_On.na						:= GVL.IOME.C_Mn_Ct.na;
//-------SIGNAL -> S_Mn_Ct Max: 1 Min: 0 Def: 0 Resolution: 1 Offset: 0
GVL.IOVD.S_Mn_Ct.v							:= GVL.SY.S_ECU_Rdy AND NOT GVL.IOVD.S_Mn_Ct.e AND NOT GVL.IOVD.S_Mn_Ct.na;
GVL.IOVD.S_Mn_Ct.x							:= GVL.IIME.S_Mn_Ct.x;
GVL.IOVD.S_Mn_Ct.e							:= GVL.IIME.S_Mn_Ct.e;
GVL.IOVD.S_Mn_Ct.na							:= GVL.IIME.S_Mn_Ct.na;
//-------SIGNAL -> C_Prechrg_Ct_On Max: 1 Min: 0 Def: 0 Resolution: 1 Offset: 0
GVL.IOVD.C_Prechrg_Ct_On.v					:= FALSE;
GVL.IOVD.C_Prechrg_Ct_On.x					:= FALSE;
GVL.IOVD.C_Prechrg_Ct_On.e					:= FALSE;
GVL.IOVD.C_Prechrg_Ct_On.na					:= FALSE;
//-------SIGNAL -> S_Prechrg_Ct Max: 1 Min: 0 Def: 0 Resolution: 1 Offset: 0
GVL.IOVD.S_Prechrg_Ct.v						:= GVL.SY.S_ECU_Rdy AND NOT GVL.IOVD.S_Prechrg_Ct.e AND NOT GVL.IOVD.S_Prechrg_Ct.na;
GVL.IOVD.S_Prechrg_Ct.x						:= GVL.IIPT.S_Prechrg_Ct_Act.x;
GVL.IOVD.S_Prechrg_Ct.e						:= GVL.IIPT.S_Prechrg_Ct_Act.e;
GVL.IOVD.S_Prechrg_Ct.na					:= GVL.IIPT.S_Prechrg_Ct_Act.na;
//-------SIGNAL -> S_ER_HV Max: 1 Min: 0 Def: 0 Resolution: 1 Offset: 0
GVL.IOVD.S_ER_HV.v							:= GVL.SY.S_ECU_Rdy AND NOT GVL.IOVD.S_ER_HV.e AND NOT GVL.IOVD.S_ER_HV.na;
GVL.IOVD.S_ER_HV.x							:= GVL.ME.S_Err_HV_Amb OR GVL.ME.S_Err_HV_Red;
GVL.IOVD.S_ER_HV.e							:= FALSE;
GVL.IOVD.S_ER_HV.na							:= FALSE;
//-------SIGNAL -> S_ER_Mn_Ct Max: 1 Min: 0 Def: 0 Resolution: 1 Offset: 0
GVL.IOVD.S_ER_Mn_Ct.v						:= FALSE;	// KULLANILMIYOR
GVL.IOVD.S_ER_Mn_Ct.x						:= FALSE;	// KULLANILMIYOR
GVL.IOVD.S_ER_Mn_Ct.e						:= FALSE;	// KULLANILMIYOR
GVL.IOVD.S_ER_Mn_Ct.na						:= FALSE;	// KULLANILMIYOR
//-------SIGNAL -> S_ER_Prechrg_Ct Max: 1 Min: 0 Def: 0 Resolution: 1 Offset: 0
GVL.IOVD.S_ER_Prechrg_Ct.v					:= FALSE;
GVL.IOVD.S_ER_Prechrg_Ct.x					:= FALSE;
GVL.IOVD.S_ER_Prechrg_Ct.e					:= FALSE;
GVL.IOVD.S_ER_Prechrg_Ct.na					:= FALSE;
//-------SIGNAL -> S_Hv_On Max: 1 Min: 0 Def: 0 Resolution: 1 Offset: 0
GVL.IOVD.S_Hv_On.v							:= GVL.SY.S_ECU_Rdy AND NOT GVL.IOVD.S_Hv_On.e AND NOT GVL.IOVD.S_Hv_On.na;
GVL.IOVD.S_Hv_On.x							:= GVL.ME.S_HV_On;
GVL.IOVD.S_Hv_On.e							:= FALSE;
GVL.IOVD.S_Hv_On.na							:= FALSE;	  
//-------SIGNAL -> S_HV_HVAC_En Max: 1 Min: 0 Def: 0 Resolution: 1 Offset: 0
GVL.IOVD.S_HV_HVAC_En.v						:= GVL.SY.S_ECU_Rdy AND NOT GVL.IOVD.S_HV_HVAC_En.e AND NOT GVL.IOVD.S_HV_HVAC_En.na;
GVL.IOVD.S_HV_HVAC_En.x						:= GVL.ME.C_HVAC_En;
GVL.IOVD.S_HV_HVAC_En.e						:= FALSE;
GVL.IOVD.S_HV_HVAC_En.na					:= FALSE;
{endregion}
//-----------------------------------------------------------------------------------------------------------------------------
//-----------------------------------------------------------------------------------------------------------------------------
//MESSAGE------
{region " User Area : TCU_Trolleybus_Durum- ID:460"}

